LIN {X 0,Y 439.389,Z 296.378,A -85,B 0,C 180,E1 -8958.743,E2 -8958.743} C_VEL
LIN {X 0,Y 439.369,Z 296.379,A -85,B 0,C 180,E1 -8961.609,E2 -8961.609} C_VEL
LIN {X 0,Y 439.4,Z 296.377,A -85,B 0,C 180,E1 -8964.844,E2 -8964.844} C_VEL
LIN {X 0,Y 439.373,Z 296.38,A -85,B 0,C 180,E1 -8968.139,E2 -8968.139} C_VEL
LIN {X 0,Y 439.399,Z 296.377,A -85,B 0,C 180,E1 -8971.606,E2 -8971.606} C_VEL
LIN {X 0,Y 439.372,Z 296.374,A -85,B 0,C 180,E1 -8974.413,E2 -8974.413} C_VEL
LIN {X 0,Y 439.364,Z 296.375,A -85,B 0,C 180,E1 -8977.424,E2 -8977.424} C_VEL
LIN {X 0,Y 439.441,Z 296.372,A -85,B 0,C 180,E1 -8980.663,E2 -8980.663} C_VEL
LIN {X 0,Y 439.463,Z 296.365,A -85,B 0,C 180,E1 -8984.224,E2 -8984.224} C_VEL
LIN {X 0,Y 439.484,Z 296.358,A -85,B 0,C 180,E1 -8988.001,E2 -8988.001} C_VEL
LIN {X 0,Y 439.503,Z 296.366,A -85,B 0,C 180,E1 -8991.725,E2 -8991.725} C_VEL
LIN {X 0,Y 439.603,Z 296.341,A -85,B 0,C 180,E1 -8994.495,E2 -8994.495} C_VEL
LIN {X 0,Y 439.635,Z 296.346,A -85,B 0,C 180,E1 -8998.168,E2 -8998.168} C_VEL
LIN {X 0,Y 439.763,Z 296.319,A -85,B 0,C 180,E1 -9000,E2 -9000} C_VEL
LIN {X 0,Y 439.628,Z 296.347,A -85,B 0,C 180,E1 -9002.749,E2 -9002.749} C_VEL
LIN {X 0,Y 439.595,Z 296.344,A -85,B 0,C 180,E1 -9006.425,E2 -9006.425} C_VEL
LIN {X 0,Y 439.497,Z 296.361,A -85,B 0,C 180,E1 -9009.202,E2 -9009.202} C_VEL
LIN {X 0,Y 439.465,Z 296.366,A -85,B 0,C 180,E1 -9012.938,E2 -9012.938} C_VEL
LIN {X 0,Y 439.446,Z 296.36,A -85,B 0,C 180,E1 -9016.348,E2 -9016.348} C_VEL
LIN {X 0,Y 439.402,Z 296.376,A -85,B 0,C 180,E1 -9019.626,E2 -9019.626} C_VEL
LIN {X 0,Y 439.363,Z 296.377,A -85,B 0,C 180,E1 -9022.575,E2 -9022.575} C_VEL
LIN {X 0,Y 439.371,Z 296.374,A -85,B 0,C 180,E1 -9025.587,E2 -9025.587} C_VEL
LIN {X 0,Y 439.396,Z 296.38,A -85,B 0,C 180,E1 -9028.675,E2 -9028.675} C_VEL
LIN {X 0,Y 439.37,Z 296.382,A -85,B 0,C 180,E1 -9032.03,E2 -9032.03} C_VEL
LIN {X 0,Y 439.392,Z 296.38,A -85,B 0,C 180,E1 -9035.34,E2 -9035.34} C_VEL
LIN {X 0,Y 439.368,Z 296.383,A -85,B 0,C 180,E1 -9038.596,E2 -9038.596} C_VEL
LIN {X 0,Y 439.388,Z 296.377,A -85,B 0,C 180,E1 -9041.257,E2 -9041.257} C_VEL
LIN {X 0,Y 439.398,Z 296.371,A -85,B 0,C 180,E1 -9044.73,E2 -9044.73} C_VEL
LIN {X 0,Y 439.405,Z 296.513,A -85,B 0,C 180,E1 -9045.613,E2 -9045.613} C_VEL
LIN {X 0,Y 442.197,Z 307.685,A -85,B 0,C 180,E1 -9048.888,E2 -9048.888} C_VEL
LIN {X 0,Y 445.159,Z 319.506,A -85,B 0,C 180,E1 -9052.127,E2 -9052.127} C_VEL
LIN {X 0,Y 446.738,Z 326.126,A -85,B 0,C 180,E1 -9053.847,E2 -9053.847} C_VEL
LIN {X 0,Y 445.922,Z 334.334,A -85,B 0,C 180,E1 -9055.706,E2 -9055.706} C_VEL
LIN {X 0,Y 444.194,Z 349.593,A -85,B 0,C 180,E1 -9059.055,E2 -9059.055} C_VEL
LIN {X 0,Y 442.682,Z 366.195,A -85,B 0,C 180,E1 -9062.587,E2 -9062.587} C_VEL
LIN {X 0,Y 441.378,Z 382.993,A -85,B 0,C 180,E1 -9066.044,E2 -9066.044} C_VEL
LIN {X 0,Y 441.077,Z 387.978,A -85,B 0,C 180,E1 -9067.06,E2 -9067.06} C_VEL
LIN {X 0,Y 444.313,Z 406.784,A -85,B 0,C 180,E1 -9067.609,E2 -9067.609} C_VEL
LIN {X 0,Y 446.055,Z 420.769,A -85,B 0,C 180,E1 -9068.139,E2 -9068.139} C_VEL
LIN {X 0,Y 445.379,Z 435.92,A -85,B 0,C 180,E1 -9068.78,E2 -9068.78} C_VEL
LIN {X 0,Y 444.458,Z 449.486,A -85,B 0,C 180,E1 -9069.522,E2 -9069.522} C_VEL
LIN {X 0,Y 443.472,Z 462.876,A -85,B 0,C 180,E1 -9070.441,E2 -9070.441} C_VEL
LIN {X 0,Y 442.399,Z 476.497,A -85,B 0,C 180,E1 -9071.595,E2 -9071.595} C_VEL
LIN {X 0,Y 441.444,Z 489.247,A -85,B 0,C 180,E1 -9072.916,E2 -9072.916} C_VEL
LIN {X 0,Y 440.591,Z 500.172,A -85,B 0,C 180,E1 -9074.266,E2 -9074.266} C_VEL
LIN {X 0,Y 439.816,Z 511.139,A -85,B 0,C 180,E1 -9075.896,E2 -9075.896} C_VEL
LIN {X 0,Y 439.272,Z 519.671,A -85,B 0,C 180,E1 -9077.408,E2 -9077.408} C_VEL
LIN {X 0,Y 439.019,Z 526.835,A -85,B 0,C 180,E1 -9078.925,E2 -9078.925} C_VEL
LIN {X 0,Y 438.661,Z 534.097,A -85,B 0,C 180,E1 -9080.781,E2 -9080.781} C_VEL
LIN {X 0,Y 438.597,Z 539.824,A -85,B 0,C 180,E1 -9082.635,E2 -9082.635} C_VEL
LIN {X 0,Y 438.6,Z 544.148,A -85,B 0,C 180,E1 -9084.483,E2 -9084.483} C_VEL
LIN {X 0,Y 438.618,Z 547.18,A -85,B 0,C 180,E1 -9086.325,E2 -9086.325} C_VEL
LIN {X 0,Y 438.595,Z 548.988,A -85,B 0,C 180,E1 -9088.164,E2 -9088.164} C_VEL
LIN {X 0,Y 438.532,Z 549.6,A -85,B 0,C 180,E1 -9090,E2 -9090} C_VEL
LIN {X 0,Y 438.586,Z 548.989,A -85,B 0,C 180,E1 -9091.837,E2 -9091.837} C_VEL
LIN {X 0,Y 438.643,Z 547.187,A -85,B 0,C 180,E1 -9093.675,E2 -9093.675} C_VEL
LIN {X 0,Y 438.639,Z 544.152,A -85,B 0,C 180,E1 -9095.517,E2 -9095.517} C_VEL
LIN {X 0,Y 438.607,Z 539.818,A -85,B 0,C 180,E1 -9097.365,E2 -9097.365} C_VEL
LIN {X 0,Y 438.683,Z 534.095,A -85,B 0,C 180,E1 -9099.219,E2 -9099.219} C_VEL
LIN {X 0,Y 439.041,Z 526.837,A -85,B 0,C 180,E1 -9101.075,E2 -9101.075} C_VEL
LIN {X 0,Y 439.284,Z 519.632,A -85,B 0,C 180,E1 -9102.598,E2 -9102.598} C_VEL
LIN {X 0,Y 439.825,Z 511.129,A -85,B 0,C 180,E1 -9104.104,E2 -9104.104} C_VEL
LIN {X 0,Y 440.431,Z 501.812,A -85,B 0,C 180,E1 -9105.503,E2 -9105.503} C_VEL
LIN {X 0,Y 441.354,Z 490.463,A -85,B 0,C 180,E1 -9106.939,E2 -9106.939} C_VEL
LIN {X 0,Y 442.217,Z 478.837,A -85,B 0,C 180,E1 -9108.174,E2 -9108.174} C_VEL
LIN {X 0,Y 443.281,Z 465.732,A -85,B 0,C 180,E1 -9109.327,E2 -9109.327} C_VEL
LIN {X 0,Y 444.232,Z 453.008,A -85,B 0,C 180,E1 -9110.248,E2 -9110.248} C_VEL
LIN {X 0,Y 445.224,Z 438.12,A -85,B 0,C 180,E1 -9111.107,E2 -9111.107} C_VEL
LIN {X 0,Y 446.061,Z 422.741,A -85,B 0,C 180,E1 -9111.779,E2 -9111.779} C_VEL
LIN {X 0,Y 445.392,Z 415.694,A -85,B 0,C 180,E1 -9112.067,E2 -9112.067} C_VEL
LIN {X 0,Y 443.655,Z 400.689,A -85,B 0,C 180,E1 -9112.565,E2 -9112.565} C_VEL
LIN {X 0,Y 440.811,Z 384.764,A -85,B 0,C 180,E1 -9113.017,E2 -9113.017} C_VEL
LIN {X 0,Y 441.759,Z 369.337,A -85,B 0,C 180,E1 -9116.199,E2 -9116.199} C_VEL
LIN {X 0,Y 443.194,Z 354.719,A -85,B 0,C 180,E1 -9119.445,E2 -9119.445} C_VEL
LIN {X 0,Y 444.848,Z 342.227,A -85,B 0,C 180,E1 -9122.49,E2 -9122.49} C_VEL
LIN {X 0,Y 447.211,Z 331.063,A -85,B 0,C 180,E1 -9125.554,E2 -9125.554} C_VEL
LIN {X 0,Y 447.513,Z 329.378,A -85,B 0,C 180,E1 -9126.081,E2 -9126.081} C_VEL
LIN {X 0,Y 446.545,Z 324.729,A -85,B 0,C 180,E1 -9127.866,E2 -9127.866} C_VEL
LIN {X 0,Y 445.197,Z 319.492,A -85,B 0,C 180,E1 -9130.334,E2 -9130.334} C_VEL
LIN {X 0,Y 444.029,Z 315.439,A -85,B 0,C 180,E1 -9132.891,E2 -9132.891} C_VEL
LIN {X 0,Y 443.498,Z 313.503,A -85,B 0,C 180,E1 -9134.512,E2 -9134.512} C_VEL
LIN {X 0,Y 442.845,Z 311.488,A -85,B 0,C 180,E1 -9136.968,E2 -9136.968} C_VEL
LIN {X 0,Y 442.349,Z 310.332,A -85,B 0,C 180,E1 -9139.696,E2 -9139.696} C_VEL
LIN {X 0,Y 442.022,Z 310.093,A -85,B 0,C 180,E1 -9142.654,E2 -9142.654} C_VEL
LIN {X 0,Y 441.698,Z 310.52,A -85,B 0,C 180,E1 -9145.054,E2 -9145.054} C_VEL
LIN {X 0,Y 441.188,Z 311.719,A -85,B 0,C 180,E1 -9148.286,E2 -9148.286} C_VEL
LIN {X 0,Y 440.867,Z 313.275,A -85,B 0,C 180,E1 -9151.43,E2 -9151.43} C_VEL
LIN {X 0,Y 440.617,Z 315.071,A -85,B 0,C 180,E1 -9154.491,E2 -9154.491} C_VEL
LIN {X 0,Y 440.408,Z 317.208,A -85,B 0,C 180,E1 -9157.754,E2 -9157.754} C_VEL
LIN {X 0,Y 440.22,Z 319.148,A -85,B 0,C 180,E1 -9160.412,E2 -9160.412} C_VEL
LIN {X 0,Y 440.105,Z 320.778,A -85,B 0,C 180,E1 -9162.575,E2 -9162.575} C_VEL
LIN {X 0,Y 445.525,Z 334.754,A -85,B 0,C 180,E1 -9163.565,E2 -9163.565} C_VEL
LIN {X 0,Y 445.75,Z 336.95,A -85,B 0,C 180,E1 -9163.695,E2 -9163.695} C_VEL
LIN {X 0,Y 445.108,Z 349.492,A -85,B 0,C 180,E1 -9164.43,E2 -9164.43} C_VEL
LIN {X 0,Y 444.362,Z 361.649,A -85,B 0,C 180,E1 -9165.342,E2 -9165.342} C_VEL
LIN {X 0,Y 443.551,Z 372.693,A -85,B 0,C 180,E1 -9166.368,E2 -9166.368} C_VEL
LIN {X 0,Y 442.7,Z 383.554,A -85,B 0,C 180,E1 -9167.625,E2 -9167.625} C_VEL
LIN {X 0,Y 441.92,Z 393.206,A -85,B 0,C 180,E1 -9168.998,E2 -9168.998} C_VEL
LIN {X 0,Y 441.307,Z 400.935,A -85,B 0,C 180,E1 -9170.374,E2 -9170.374} C_VEL
LIN {X 0,Y 440.756,Z 407.201,A -85,B 0,C 180,E1 -9171.749,E2 -9171.749} C_VEL
LIN {X 0,Y 440.312,Z 412.208,A -85,B 0,C 180,E1 -9173.125,E2 -9173.125} C_VEL
LIN {X 0,Y 439.832,Z 416.126,A -85,B 0,C 180,E1 -9174.499,E2 -9174.499} C_VEL
LIN {X 0,Y 439.752,Z 418.15,A -85,B 0,C 180,E1 -9175.417,E2 -9175.417} C_VEL
LIN {X 0,Y 439.742,Z 419.744,A -85,B 0,C 180,E1 -9176.335,E2 -9176.335} C_VEL
LIN {X 0,Y 439.548,Z 420.923,A -85,B 0,C 180,E1 -9177.251,E2 -9177.251} C_VEL
LIN {X 0,Y 439.327,Z 422.086,A -85,B 0,C 180,E1 -9179.083,E2 -9179.083} C_VEL
LIN {X 0,Y 439.293,Z 422.079,A -85,B 0,C 180,E1 -9180,E2 -9180} C_VEL
LIN {X 0,Y 439.301,Z 421.639,A -85,B 0,C 180,E1 -9180.917,E2 -9180.917} C_VEL
LIN {X 0,Y 439.155,Z 419.614,A -85,B 0,C 180,E1 -9182.752,E2 -9182.752} C_VEL
LIN {X 0,Y 439.293,Z 416.979,A -85,B 0,C 180,E1 -9184.129,E2 -9184.129} C_VEL
LIN {X 0,Y 439.475,Z 413.358,A -85,B 0,C 180,E1 -9185.506,E2 -9185.506} C_VEL
LIN {X 0,Y 439.772,Z 408.664,A -85,B 0,C 180,E1 -9186.884,E2 -9186.884} C_VEL
LIN {X 0,Y 440.131,Z 401.693,A -85,B 0,C 180,E1 -9188.494,E2 -9188.494} C_VEL
LIN {X 0,Y 440.5,Z 394.142,A -85,B 0,C 180,E1 -9189.876,E2 -9189.876} C_VEL
LIN {X 0,Y 440.906,Z 384.875,A -85,B 0,C 180,E1 -9191.26,E2 -9191.26} C_VEL
LIN {X 0,Y 441.518,Z 375.436,A -85,B 0,C 180,E1 -9192.409,E2 -9192.409} C_VEL
LIN {X 0,Y 442.075,Z 363.806,A -85,B 0,C 180,E1 -9193.562,E2 -9193.562} C_VEL
LIN {X 0,Y 442.644,Z 351.293,A -85,B 0,C 180,E1 -9194.557,E2 -9194.557} C_VEL
LIN {X 0,Y 443.145,Z 338.462,A -85,B 0,C 180,E1 -9195.346,E2 -9195.346} C_VEL
LIN {X 0,Y 443.417,Z 330.363,A -85,B 0,C 180,E1 -9195.749,E2 -9195.749} C_VEL
LIN {X 0,Y 439.904,Z 316.829,A -85,B 0,C 180,E1 -9196.403,E2 -9196.403} C_VEL
LIN {X 0,Y 438.766,Z 312.57,A -85,B 0,C 180,E1 -9196.589,E2 -9196.589} C_VEL
LIN {X 0,Y 438.819,Z 309.161,A -85,B 0,C 180,E1 -9199.654,E2 -9199.654} C_VEL
LIN {X 0,Y 438.808,Z 305.945,A -85,B 0,C 180,E1 -9202.606,E2 -9202.606} C_VEL
LIN {X 0,Y 438.815,Z 302.707,A -85,B 0,C 180,E1 -9205.622,E2 -9205.622} C_VEL
LIN {X 0,Y 438.855,Z 299.441,A -85,B 0,C 180,E1 -9208.714,E2 -9208.714} C_VEL
LIN {X 0,Y 438.863,Z 297.207,A -85,B 0,C 180,E1 -9210.827,E2 -9210.827} C_VEL
LIN {X 0,Y 438.924,Z 296.439,A -85,B 0,C 180,E1 -9211.936,E2 -9211.936} C_VEL
LIN {X 0,Y 439.305,Z 296.391,A -85,B 0,C 180,E1 -9215.323,E2 -9215.323} C_VEL
LIN {X 0,Y 439.385,Z 296.379,A -85,B 0,C 180,E1 -9218.595,E2 -9218.595} C_VEL
LIN {X 0,Y 439.391,Z 296.374,A -85,B 0,C 180,E1 -9221.257,E2 -9221.257} C_VEL
LIN {X 0,Y 439.401,Z 296.375,A -85,B 0,C 180,E1 -9224.729,E2 -9224.729} C_VEL
LIN {X 0,Y 439.342,Z 296.387,A -85,B 0,C 180,E1 -9228.305,E2 -9228.305} C_VEL
LIN {X 0,Y 439.405,Z 296.687,A -85,B 0,C 180,E1 -9228.741,E2 -9228.741} C_VEL
LIN {X 0,Y 439.466,Z 300.718,A -85,B 0,C 180,E1 -9231.593,E2 -9231.593} C_VEL
LIN {X 0,Y 439.393,Z 305.155,A -85,B 0,C 180,E1 -9234.843,E2 -9234.843} C_VEL
LIN {X 0,Y 439.321,Z 309.591,A -85,B 0,C 180,E1 -9238.135,E2 -9238.135} C_VEL
LIN {X 0,Y 439.259,Z 313.984,A -85,B 0,C 180,E1 -9241.315,E2 -9241.315} C_VEL
LIN {X 0,Y 439.204,Z 318.505,A -85,B 0,C 180,E1 -9244.402,E2 -9244.402} C_VEL
LIN {X 0,Y 439.232,Z 322.302,A -85,B 0,C 180,E1 -9246.82,E2 -9246.82} C_VEL
LIN {X 0,Y 445.434,Z 339.613,A -85,B 0,C 180,E1 -9247.592,E2 -9247.592} C_VEL
LIN {X 0,Y 447.746,Z 347.503,A -85,B 0,C 180,E1 -9247.99,E2 -9247.99} C_VEL
LIN {X 0,Y 447.094,Z 362.755,A -85,B 0,C 180,E1 -9248.636,E2 -9248.636} C_VEL
LIN {X 0,Y 446.37,Z 375.925,A -85,B 0,C 180,E1 -9249.372,E2 -9249.372} C_VEL
LIN {X 0,Y 445.502,Z 389.149,A -85,B 0,C 180,E1 -9250.293,E2 -9250.293} C_VEL
LIN {X 0,Y 444.516,Z 401.345,A -85,B 0,C 180,E1 -9251.327,E2 -9251.327} C_VEL
LIN {X 0,Y 443.447,Z 413.714,A -85,B 0,C 180,E1 -9252.594,E2 -9252.594} C_VEL
LIN {X 0,Y 442.525,Z 424.069,A -85,B 0,C 180,E1 -9253.863,E2 -9253.863} C_VEL
LIN {X 0,Y 441.646,Z 433.644,A -85,B 0,C 180,E1 -9255.249,E2 -9255.249} C_VEL
LIN {X 0,Y 440.798,Z 442.36,A -85,B 0,C 180,E1 -9256.741,E2 -9256.741} C_VEL
LIN {X 0,Y 440.645,Z 444.982,A -85,B 0,C 180,E1 -9257.254,E2 -9257.254} C_VEL
LIN {X 0,Y 439.716,Z 448.238,A -85,B 0,C 180,E1 -9257.885,E2 -9257.885} C_VEL
LIN {X 0,Y 436.468,Z 453.328,A -85,B 0,C 180,E1 -9258.914,E2 -9258.914} C_VEL
LIN {X 0,Y 433.252,Z 457.905,A -85,B 0,C 180,E1 -9259.995,E2 -9259.995} C_VEL
LIN {X 0,Y 432.389,Z 460.347,A -85,B 0,C 180,E1 -9260.699,E2 -9260.699} C_VEL
LIN {X 0,Y 431.991,Z 465.553,A -85,B 0,C 180,E1 -9262.521,E2 -9262.521} C_VEL
LIN {X 0,Y 431.657,Z 469.62,A -85,B 0,C 180,E1 -9264.394,E2 -9264.394} C_VEL
LIN {X 0,Y 431.642,Z 472.459,A -85,B 0,C 180,E1 -9266.266,E2 -9266.266} C_VEL
LIN {X 0,Y 431.424,Z 474.18,A -85,B 0,C 180,E1 -9268.133,E2 -9268.133} C_VEL
LIN {X 0,Y 431.308,Z 474.781,A -85,B 0,C 180,E1 -9270,E2 -9270} C_VEL
LIN {X 0,Y 431.423,Z 474.223,A -85,B 0,C 180,E1 -9271.867,E2 -9271.867} C_VEL
LIN {X 0,Y 431.63,Z 472.562,A -85,B 0,C 180,E1 -9273.734,E2 -9273.734} C_VEL
LIN {X 0,Y 431.653,Z 469.789,A -85,B 0,C 180,E1 -9275.606,E2 -9275.606} C_VEL
LIN {X 0,Y 432.015,Z 465.79,A -85,B 0,C 180,E1 -9277.478,E2 -9277.478} C_VEL
LIN {X 0,Y 432.385,Z 460.486,A -85,B 0,C 180,E1 -9279.354,E2 -9279.354} C_VEL
LIN {X 0,Y 432.988,Z 453.71,A -85,B 0,C 180,E1 -9281.231,E2 -9281.231} C_VEL
LIN {X 0,Y 433.668,Z 446.448,A -85,B 0,C 180,E1 -9282.875,E2 -9282.875} C_VEL
LIN {X 0,Y 434.451,Z 437.686,A -85,B 0,C 180,E1 -9284.521,E2 -9284.521} C_VEL
LIN {X 0,Y 435.515,Z 427.072,A -85,B 0,C 180,E1 -9286.163,E2 -9286.163} C_VEL
LIN {X 0,Y 436.547,Z 416.162,A -85,B 0,C 180,E1 -9287.569,E2 -9287.569} C_VEL
LIN {X 0,Y 437.654,Z 404.17,A -85,B 0,C 180,E1 -9288.855,E2 -9288.855} C_VEL
LIN {X 0,Y 438.74,Z 390.926,A -85,B 0,C 180,E1 -9290.023,E2 -9290.023} C_VEL
LIN {X 0,Y 439.728,Z 377.966,A -85,B 0,C 180,E1 -9290.953,E2 -9290.953} C_VEL
LIN {X 0,Y 440.589,Z 363.194,A -85,B 0,C 180,E1 -9291.797,E2 -9291.797} C_VEL
LIN {X 0,Y 441.033,Z 348.463,A -85,B 0,C 180,E1 -9292.444,E2 -9292.444} C_VEL
LIN {X 0,Y 436.308,Z 334.096,A -85,B 0,C 180,E1 -9293.182,E2 -9293.182} C_VEL
LIN {X 0,Y 432.227,Z 322.877,A -85,B 0,C 180,E1 -9293.677,E2 -9293.677} C_VEL
LIN {X 0,Y 432.245,Z 317.598,A -85,B 0,C 180,E1 -9297.082,E2 -9297.082} C_VEL
LIN {X 0,Y 432.289,Z 313.042,A -85,B 0,C 180,E1 -9300.264,E2 -9300.264} C_VEL
LIN {X 0,Y 432.357,Z 307.993,A -85,B 0,C 180,E1 -9304.003,E2 -9304.003} C_VEL
LIN {X 0,Y 432.41,Z 303.622,A -85,B 0,C 180,E1 -9307.212,E2 -9307.212} C_VEL
LIN {X 0,Y 432.456,Z 299.531,A -85,B 0,C 180,E1 -9310.198,E2 -9310.198} C_VEL
LIN {X 0,Y 432.31,Z 297.266,A -85,B 0,C 180,E1 -9311.8,E2 -9311.8} C_VEL
LIN {X 0,Y 432.333,Z 297.26,A -85,B 0,C 180,E1 -9314.347,E2 -9314.347} C_VEL
LIN {X 0,Y 432.321,Z 297.262,A -85,B 0,C 180,E1 -9317.015,E2 -9317.015} C_VEL
LIN {X 0,Y 432.333,Z 297.258,A -85,B 0,C 180,E1 -9319.821,E2 -9319.821} C_VEL
LIN {X 0,Y 432.306,Z 297.26,A -85,B 0,C 180,E1 -9323.022,E2 -9323.022} C_VEL
LIN {X 0,Y 432.36,Z 297.25,A -85,B 0,C 180,E1 -9325.996,E2 -9325.996} C_VEL
LIN {X 0,Y 432.346,Z 297.251,A -85,B 0,C 180,E1 -9329.49,E2 -9329.49} C_VEL
LIN {X 0,Y 432.327,Z 297.26,A -85,B 0,C 180,E1 -9331.873,E2 -9331.873} C_VEL
LIN {X 0,Y 432.376,Z 297.253,A -85,B 0,C 180,E1 -9335.539,E2 -9335.539} C_VEL
LIN {X 0,Y 432.35,Z 297.251,A -85,B 0,C 180,E1 -9339.046,E2 -9339.046} C_VEL
LIN {X 0,Y 432.358,Z 297.249,A -85,B 0,C 180,E1 -9342.01,E2 -9342.01} C_VEL
LIN {X 0,Y 432.397,Z 297.247,A -85,B 0,C 180,E1 -9344.926,E2 -9344.926} C_VEL
LIN {X 0,Y 432.46,Z 297.232,A -85,B 0,C 180,E1 -9347.803,E2 -9347.803} C_VEL
LIN {X 0,Y 432.463,Z 297.242,A -85,B 0,C 180,E1 -9351.59,E2 -9351.59} C_VEL
LIN {X 0,Y 432.576,Z 297.215,A -85,B 0,C 180,E1 -9354.406,E2 -9354.406} C_VEL
LIN {X 0,Y 432.604,Z 297.221,A -85,B 0,C 180,E1 -9358.138,E2 -9358.138} C_VEL
LIN {X 0,Y 432.733,Z 297.194,A -85,B 0,C 180,E1 -9360,E2 -9360} C_VEL
LIN {X 0,Y 432.579,Z 297.225,A -85,B 0,C 180,E1 -9362.794,E2 -9362.794} C_VEL
LIN {X 0,Y 432.547,Z 297.223,A -85,B 0,C 180,E1 -9366.531,E2 -9366.531} C_VEL
LIN {X 0,Y 432.441,Z 297.24,A -85,B 0,C 180,E1 -9369.353,E2 -9369.353} C_VEL
LIN {X 0,Y 432.431,Z 297.242,A -85,B 0,C 180,E1 -9372.803,E2 -9372.803} C_VEL
LIN {X 0,Y 432.411,Z 297.236,A -85,B 0,C 180,E1 -9376.478,E2 -9376.478} C_VEL
LIN {X 0,Y 432.339,Z 297.258,A -85,B 0,C 180,E1 -9379.96,E2 -9379.96} C_VEL
LIN {X 0,Y 432.316,Z 297.255,A -85,B 0,C 180,E1 -9382.964,E2 -9382.964} C_VEL
LIN {X 0,Y 432.333,Z 297.258,A -85,B 0,C 180,E1 -9385.002,E2 -9385.002} C_VEL
LIN {X 0,Y 432.342,Z 297.253,A -85,B 0,C 180,E1 -9388.126,E2 -9388.126} C_VEL
LIN {X 0,Y 432.32,Z 297.258,A -85,B 0,C 180,E1 -9391.346,E2 -9391.346} C_VEL
LIN {X 0,Y 432.338,Z 297.255,A -85,B 0,C 180,E1 -9394.677,E2 -9394.677} C_VEL
LIN {X 0,Y 432.331,Z 297.259,A -85,B 0,C 180,E1 -9398.15,E2 -9398.15} C_VEL
LIN {X 0,Y 432.332,Z 297.256,A -85,B 0,C 180,E1 -9401.602,E2 -9401.602} C_VEL
LIN {X 0,Y 432.369,Z 297.359,A -85,B 0,C 180,E1 -9405.08,E2 -9405.08} C_VEL
LIN {X 0,Y 435.202,Z 308.884,A -85,B 0,C 180,E1 -9408.54,E2 -9408.54} C_VEL
LIN {X 0,Y 437.783,Z 319.165,A -85,B 0,C 180,E1 -9411.427,E2 -9411.427} C_VEL
LIN {X 0,Y 439.885,Z 327.94,A -85,B 0,C 180,E1 -9413.762,E2 -9413.762} C_VEL
LIN {X 0,Y 439.027,Z 336.115,A -85,B 0,C 180,E1 -9415.647,E2 -9415.647} C_VEL
LIN {X 0,Y 437.106,Z 352.498,A -85,B 0,C 180,E1 -9419.304,E2 -9419.304} C_VEL
LIN {X 0,Y 435.528,Z 368.731,A -85,B 0,C 180,E1 -9422.825,E2 -9422.825} C_VEL
LIN {X 0,Y 434.297,Z 384.479,A -85,B 0,C 180,E1 -9426.136,E2 -9426.136} C_VEL
LIN {X 0,Y 434.111,Z 387.031,A -85,B 0,C 180,E1 -9426.663,E2 -9426.663} C_VEL
LIN {X 0,Y 437.608,Z 406.962,A -85,B 0,C 180,E1 -9427.267,E2 -9427.267} C_VEL
LIN {X 0,Y 439.369,Z 421.804,A -85,B 0,C 180,E1 -9427.854,E2 -9427.854} C_VEL
LIN {X 0,Y 438.658,Z 436.472,A -85,B 0,C 180,E1 -9428.501,E2 -9428.501} C_VEL
LIN {X 0,Y 437.619,Z 450.671,A -85,B 0,C 180,E1 -9429.31,E2 -9429.31} C_VEL
LIN {X 0,Y 436.582,Z 463.723,A -85,B 0,C 180,E1 -9430.242,E2 -9430.242} C_VEL
LIN {X 0,Y 435.473,Z 477.078,A -85,B 0,C 180,E1 -9431.413,E2 -9431.413} C_VEL
LIN {X 0,Y 434.589,Z 488.148,A -85,B 0,C 180,E1 -9432.578,E2 -9432.578} C_VEL
LIN {X 0,Y 433.658,Z 499.56,A -85,B 0,C 180,E1 -9434.008,E2 -9434.008} C_VEL
LIN {X 0,Y 432.803,Z 510.523,A -85,B 0,C 180,E1 -9435.663,E2 -9435.663} C_VEL
LIN {X 0,Y 432.21,Z 519.683,A -85,B 0,C 180,E1 -9437.326,E2 -9437.326} C_VEL
LIN {X 0,Y 431.875,Z 528.205,A -85,B 0,C 180,E1 -9439.214,E2 -9439.214} C_VEL
LIN {X 0,Y 431.551,Z 535.064,A -85,B 0,C 180,E1 -9441.1,E2 -9441.1} C_VEL
LIN {X 0,Y 431.515,Z 540.444,A -85,B 0,C 180,E1 -9442.984,E2 -9442.984} C_VEL
LIN {X 0,Y 431.533,Z 543.539,A -85,B 0,C 180,E1 -9444.392,E2 -9444.392} C_VEL
LIN {X 0,Y 431.549,Z 546.572,A -85,B 0,C 180,E1 -9446.265,E2 -9446.265} C_VEL
LIN {X 0,Y 431.533,Z 548.38,A -85,B 0,C 180,E1 -9448.134,E2 -9448.134} C_VEL
LIN {X 0,Y 431.461,Z 548.992,A -85,B 0,C 180,E1 -9450,E2 -9450} C_VEL
LIN {X 0,Y 431.525,Z 548.382,A -85,B 0,C 180,E1 -9451.867,E2 -9451.867} C_VEL
LIN {X 0,Y 431.577,Z 546.578,A -85,B 0,C 180,E1 -9453.735,E2 -9453.735} C_VEL
LIN {X 0,Y 431.57,Z 543.541,A -85,B 0,C 180,E1 -9455.607,E2 -9455.607} C_VEL
LIN {X 0,Y 431.527,Z 539.204,A -85,B 0,C 180,E1 -9457.487,E2 -9457.487} C_VEL
LIN {X 0,Y 431.621,Z 533.48,A -85,B 0,C 180,E1 -9459.371,E2 -9459.371} C_VEL
LIN {X 0,Y 431.949,Z 526.217,A -85,B 0,C 180,E1 -9461.259,E2 -9461.259} C_VEL
LIN {X 0,Y 432.27,Z 519.036,A -85,B 0,C 180,E1 -9462.802,E2 -9462.802} C_VEL
LIN {X 0,Y 432.813,Z 510.509,A -85,B 0,C 180,E1 -9464.337,E2 -9464.337} C_VEL
LIN {X 0,Y 433.514,Z 501.198,A -85,B 0,C 180,E1 -9465.757,E2 -9465.757} C_VEL
LIN {X 0,Y 434.402,Z 490.739,A -85,B 0,C 180,E1 -9467.11,E2 -9467.11} C_VEL
LIN {X 0,Y 435.281,Z 479.413,A -85,B 0,C 180,E1 -9468.352,E2 -9468.352} C_VEL
LIN {X 0,Y 436.39,Z 466.562,A -85,B 0,C 180,E1 -9469.523,E2 -9469.523} C_VEL
LIN {X 0,Y 437.509,Z 452.406,A -85,B 0,C 180,E1 -9470.573,E2 -9470.573} C_VEL
LIN {X 0,Y 438.566,Z 437.529,A -85,B 0,C 180,E1 -9471.443,E2 -9471.443} C_VEL
LIN {X 0,Y 439.406,Z 422.466,A -85,B 0,C 180,E1 -9472.113,E2 -9472.113} C_VEL
LIN {X 0,Y 438.021,Z 409.096,A -85,B 0,C 180,E1 -9472.649,E2 -9472.649} C_VEL
LIN {X 0,Y 435.807,Z 394.15,A -85,B 0,C 180,E1 -9473.114,E2 -9473.114} C_VEL
LIN {X 0,Y 433.881,Z 384.095,A -85,B 0,C 180,E1 -9473.4,E2 -9473.4} C_VEL
LIN {X 0,Y 434.835,Z 370.016,A -85,B 0,C 180,E1 -9476.39,E2 -9476.39} C_VEL
LIN {X 0,Y 436.288,Z 356.108,A -85,B 0,C 180,E1 -9479.557,E2 -9479.557} C_VEL
LIN {X 0,Y 437.947,Z 344.254,A -85,B 0,C 180,E1 -9482.52,E2 -9482.52} C_VEL
LIN {X 0,Y 440.259,Z 333.601,A -85,B 0,C 180,E1 -9485.499,E2 -9485.499} C_VEL
LIN {X 0,Y 440.73,Z 331.477,A -85,B 0,C 180,E1 -9486.158,E2 -9486.158} C_VEL
LIN {X 0,Y 439.842,Z 327.067,A -85,B 0,C 180,E1 -9487.883,E2 -9487.883} C_VEL
LIN {X 0,Y 438.472,Z 321.694,A -85,B 0,C 180,E1 -9490.455,E2 -9490.455} C_VEL
LIN {X 0,Y 437.565,Z 318.506,A -85,B 0,C 180,E1 -9492.423,E2 -9492.423} C_VEL
LIN {X 0,Y 436.63,Z 315.319,A -85,B 0,C 180,E1 -9495.091,E2 -9495.091} C_VEL
LIN {X 0,Y 435.941,Z 313.273,A -85,B 0,C 180,E1 -9497.867,E2 -9497.867} C_VEL
LIN {X 0,Y 435.452,Z 312.288,A -85,B 0,C 180,E1 -9500.778,E2 -9500.778} C_VEL
LIN {X 0,Y 435.131,Z 312.192,A -85,B 0,C 180,E1 -9503.302,E2 -9503.302} C_VEL
LIN {X 0,Y 434.789,Z 312.607,A -85,B 0,C 180,E1 -9505.546,E2 -9505.546} C_VEL
LIN {X 0,Y 434.246,Z 313.864,A -85,B 0,C 180,E1 -9509.068,E2 -9509.068} C_VEL
LIN {X 0,Y 433.907,Z 315.279,A -85,B 0,C 180,E1 -9511.984,E2 -9511.984} C_VEL
LIN {X 0,Y 433.654,Z 317.108,A -85,B 0,C 180,E1 -9515.171,E2 -9515.171} C_VEL
LIN {X 0,Y 433.449,Z 319.023,A -85,B 0,C 180,E1 -9518.104,E2 -9518.104} C_VEL
LIN {X 0,Y 433.236,Z 321.149,A -85,B 0,C 180,E1 -9521.068,E2 -9521.068} C_VEL
LIN {X 0,Y 433.204,Z 322.098,A -85,B 0,C 180,E1 -9522.151,E2 -9522.151} C_VEL
LIN {X 0,Y 438.344,Z 334.617,A -85,B 0,C 180,E1 -9523.078,E2 -9523.078} C_VEL
LIN {X 0,Y 439.309,Z 337.522,A -85,B 0,C 180,E1 -9523.303,E2 -9523.303} C_VEL
LIN {X 0,Y 438.617,Z 350.508,A -85,B 0,C 180,E1 -9524.084,E2 -9524.084} C_VEL
LIN {X 0,Y 437.701,Z 363.845,A -85,B 0,C 180,E1 -9525.114,E2 -9525.114} C_VEL
LIN {X 0,Y 436.891,Z 374.635,A -85,B 0,C 180,E1 -9526.156,E2 -9526.156} C_VEL
LIN {X 0,Y 435.986,Z 385.314,A -85,B 0,C 180,E1 -9527.431,E2 -9527.431} C_VEL
LIN {X 0,Y 435.115,Z 394.767,A -85,B 0,C 180,E1 -9528.824,E2 -9528.824} C_VEL
LIN {X 0,Y 434.31,Z 403.527,A -85,B 0,C 180,E1 -9530.453,E2 -9530.453} C_VEL
LIN {X 0,Y 433.868,Z 408.59,A -85,B 0,C 180,E1 -9531.617,E2 -9531.617} C_VEL
LIN {X 0,Y 433.399,Z 413.543,A -85,B 0,C 180,E1 -9533.015,E2 -9533.015} C_VEL
LIN {X 0,Y 432.882,Z 417.409,A -85,B 0,C 180,E1 -9534.41,E2 -9534.41} C_VEL
LIN {X 0,Y 432.794,Z 419.388,A -85,B 0,C 180,E1 -9535.343,E2 -9535.343} C_VEL
LIN {X 0,Y 432.757,Z 420.935,A -85,B 0,C 180,E1 -9536.276,E2 -9536.276} C_VEL
LIN {X 0,Y 432.381,Z 422.822,A -85,B 0,C 180,E1 -9538.137,E2 -9538.137} C_VEL
LIN {X 0,Y 432.313,Z 423.181,A -85,B 0,C 180,E1 -9539.069,E2 -9539.069} C_VEL
LIN {X 0,Y 432.274,Z 423.143,A -85,B 0,C 180,E1 -9540,E2 -9540} C_VEL
LIN {X 0,Y 432.281,Z 422.672,A -85,B 0,C 180,E1 -9540.932,E2 -9540.932} C_VEL
LIN {X 0,Y 432.129,Z 420.581,A -85,B 0,C 180,E1 -9542.797,E2 -9542.797} C_VEL
LIN {X 0,Y 432.278,Z 417.89,A -85,B 0,C 180,E1 -9544.196,E2 -9544.196} C_VEL
LIN {X 0,Y 432.478,Z 414.213,A -85,B 0,C 180,E1 -9545.596,E2 -9545.596} C_VEL
LIN {X 0,Y 432.782,Z 409.459,A -85,B 0,C 180,E1 -9546.996,E2 -9546.996} C_VEL
LIN {X 0,Y 433.146,Z 402.399,A -85,B 0,C 180,E1 -9548.632,E2 -9548.632} C_VEL
LIN {X 0,Y 433.554,Z 394.776,A -85,B 0,C 180,E1 -9550.036,E2 -9550.036} C_VEL
LIN {X 0,Y 433.965,Z 385.428,A -85,B 0,C 180,E1 -9551.443,E2 -9551.443} C_VEL
LIN {X 0,Y 434.685,Z 374.809,A -85,B 0,C 180,E1 -9552.726,E2 -9552.726} C_VEL
LIN {X 0,Y 435.27,Z 362.872,A -85,B 0,C 180,E1 -9553.897,E2 -9553.897} C_VEL
LIN {X 0,Y 435.839,Z 350.436,A -85,B 0,C 180,E1 -9554.865,E2 -9554.865} C_VEL
LIN {X 0,Y 436.379,Z 337.522,A -85,B 0,C 180,E1 -9555.65,E2 -9555.65} C_VEL
LIN {X 0,Y 436.556,Z 331.561,A -85,B 0,C 180,E1 -9555.948,E2 -9555.948} C_VEL
LIN {X 0,Y 432.936,Z 317.83,A -85,B 0,C 180,E1 -9556.637,E2 -9556.637} C_VEL
LIN {X 0,Y 431.731,Z 313.107,A -85,B 0,C 180,E1 -9556.85,E2 -9556.85} C_VEL
LIN {X 0,Y 431.755,Z 309.621,A -85,B 0,C 180,E1 -9559.989,E2 -9559.989} C_VEL
LIN {X 0,Y 431.76,Z 306.364,A -85,B 0,C 180,E1 -9562.996,E2 -9562.996} C_VEL
LIN {X 0,Y 431.771,Z 303.043,A -85,B 0,C 180,E1 -9566.071,E2 -9566.071} C_VEL
LIN {X 0,Y 431.811,Z 299.714,A -85,B 0,C 180,E1 -9569.227,E2 -9569.227} C_VEL
LIN {X 0,Y 431.826,Z 297.447,A -85,B 0,C 180,E1 -9571.386,E2 -9571.386} C_VEL
LIN {X 0,Y 432.192,Z 297.274,A -85,B 0,C 180,E1 -9574.691,E2 -9574.691} C_VEL
LIN {X 0,Y 432.339,Z 297.254,A -85,B 0,C 180,E1 -9578.15,E2 -9578.15} C_VEL
LIN {X 0,Y 432.335,Z 297.252,A -85,B 0,C 180,E1 -9581.602,E2 -9581.602} C_VEL
LIN {X 0,Y 432.336,Z 297.255,A -85,B 0,C 180,E1 -9584.347,E2 -9584.347} C_VEL
LIN {X 0,Y 432.301,Z 297.262,A -85,B 0,C 180,E1 -9587.019,E2 -9587.019} C_VEL
LIN {X 0,Y 432.326,Z 297.377,A -85,B 0,C 180,E1 -9588.399,E2 -9588.399} C_VEL
LIN {X 0,Y 432.427,Z 300.564,A -85,B 0,C 180,E1 -9590.665,E2 -9590.665} C_VEL
LIN {X 0,Y 432.396,Z 303.811,A -85,B 0,C 180,E1 -9593.031,E2 -9593.031} C_VEL
LIN {X 0,Y 432.33,Z 308.417,A -85,B 0,C 180,E1 -9596.447,E2 -9596.447} C_VEL
LIN {X 0,Y 432.284,Z 312.899,A -85,B 0,C 180,E1 -9599.735,E2 -9599.735} C_VEL
LIN {X 0,Y 432.222,Z 317.438,A -85,B 0,C 180,E1 -9602.916,E2 -9602.916} C_VEL
LIN {X 0,Y 432.212,Z 322.882,A -85,B 0,C 180,E1 -9606.428,E2 -9606.428} C_VEL
LIN {X 0,Y 438.221,Z 339.405,A -85,B 0,C 180,E1 -9607.179,E2 -9607.179} C_VEL
LIN {X 0,Y 441.132,Z 349.115,A -85,B 0,C 180,E1 -9607.681,E2 -9607.681} C_VEL
LIN {X 0,Y 440.511,Z 363.658,A -85,B 0,C 180,E1 -9608.317,E2 -9608.317} C_VEL
LIN {X 0,Y 439.775,Z 376.516,A -85,B 0,C 180,E1 -9609.049,E2 -9609.049} C_VEL
LIN {X 0,Y 438.866,Z 389.745,A -85,B 0,C 180,E1 -9609.983,E2 -9609.983} C_VEL
LIN {X 0,Y 437.805,Z 401.947,A -85,B 0,C 180,E1 -9611.03,E2 -9611.03} C_VEL
LIN {X 0,Y 436.699,Z 414.318,A -85,B 0,C 180,E1 -9612.316,E2 -9612.316} C_VEL
LIN {X 0,Y 435.748,Z 424.673,A -85,B 0,C 180,E1 -9613.605,E2 -9613.605} C_VEL
LIN {X 0,Y 434.811,Z 434.25,A -85,B 0,C 180,E1 -9615.012,E2 -9615.012} C_VEL
LIN {X 0,Y 433.868,Z 443.238,A -85,B 0,C 180,E1 -9616.579,E2 -9616.579} C_VEL
LIN {X 0,Y 433.188,Z 451.387,A -85,B 0,C 180,E1 -9618.299,E2 -9618.299} C_VEL
LIN {X 0,Y 432.531,Z 458.625,A -85,B 0,C 180,E1 -9620.176,E2 -9620.176} C_VEL
LIN {X 0,Y 432.389,Z 460.347,A -85,B 0,C 180,E1 -9620.699,E2 -9620.699} C_VEL
LIN {X 0,Y 431.534,Z 462.652,A -85,B 0,C 180,E1 -9621.414,E2 -9621.414} C_VEL
LIN {X 0,Y 427.001,Z 467.444,A -85,B 0,C 180,E1 -9623.049,E2 -9623.049} C_VEL
LIN {X 0,Y 424.936,Z 469.714,A -85,B 0,C 180,E1 -9624.033,E2 -9624.033} C_VEL
LIN {X 0,Y 424.602,Z 470.637,A -85,B 0,C 180,E1 -9624.549,E2 -9624.549} C_VEL
LIN {X 0,Y 424.579,Z 473.068,A -85,B 0,C 180,E1 -9626.203,E2 -9626.203} C_VEL
LIN {X 0,Y 424.373,Z 474.787,A -85,B 0,C 180,E1 -9628.102,E2 -9628.102} C_VEL
LIN {X 0,Y 424.248,Z 475.389,A -85,B 0,C 180,E1 -9630,E2 -9630} C_VEL
LIN {X 0,Y 424.372,Z 474.83,A -85,B 0,C 180,E1 -9631.898,E2 -9631.898} C_VEL
LIN {X 0,Y 424.569,Z 473.17,A -85,B 0,C 180,E1 -9633.796,E2 -9633.796} C_VEL
LIN {X 0,Y 424.604,Z 470.397,A -85,B 0,C 180,E1 -9635.699,E2 -9635.699} C_VEL
LIN {X 0,Y 424.99,Z 466.398,A -85,B 0,C 180,E1 -9637.602,E2 -9637.602} C_VEL
LIN {X 0,Y 425.394,Z 461.092,A -85,B 0,C 180,E1 -9639.509,E2 -9639.509} C_VEL
LIN {X 0,Y 426.049,Z 454.314,A -85,B 0,C 180,E1 -9641.417,E2 -9641.417} C_VEL
LIN {X 0,Y 426.762,Z 447.052,A -85,B 0,C 180,E1 -9643.087,E2 -9643.087} C_VEL
LIN {X 0,Y 427.588,Z 438.289,A -85,B 0,C 180,E1 -9644.759,E2 -9644.759} C_VEL
LIN {X 0,Y 428.704,Z 427.673,A -85,B 0,C 180,E1 -9646.427,E2 -9646.427} C_VEL
LIN {X 0,Y 429.778,Z 416.761,A -85,B 0,C 180,E1 -9647.855,E2 -9647.855} C_VEL
LIN {X 0,Y 430.964,Z 404.762,A -85,B 0,C 180,E1 -9649.159,E2 -9649.159} C_VEL
LIN {X 0,Y 432.105,Z 391.511,A -85,B 0,C 180,E1 -9650.344,E2 -9650.344} C_VEL
LIN {X 0,Y 433.138,Z 378.545,A -85,B 0,C 180,E1 -9651.288,E2 -9651.288} C_VEL
LIN {X 0,Y 434.022,Z 364.224,A -85,B 0,C 180,E1 -9652.12,E2 -9652.12} C_VEL
LIN {X 0,Y 434.513,Z 350.164,A -85,B 0,C 180,E1 -9652.754,E2 -9652.754} C_VEL
LIN {X 0,Y 429.898,Z 336.047,A -85,B 0,C 180,E1 -9653.507,E2 -9653.507} C_VEL
LIN {X 0,Y 425.205,Z 323.442,A -85,B 0,C 180,E1 -9654.095,E2 -9654.095} C_VEL
LIN {X 0,Y 425.231,Z 318.071,A -85,B 0,C 180,E1 -9657.566,E2 -9657.566} C_VEL
LIN {X 0,Y 425.271,Z 314.997,A -85,B 0,C 180,E1 -9659.721,E2 -9659.721} C_VEL
LIN {X 0,Y 425.291,Z 310.392,A -85,B 0,C 180,E1 -9663.047,E2 -9663.047} C_VEL
LIN {X 0,Y 425.339,Z 306.513,A -85,B 0,C 180,E1 -9665.939,E2 -9665.939} C_VEL
LIN {X 0,Y 425.44,Z 302.256,A -85,B 0,C 180,E1 -9669.067,E2 -9669.067} C_VEL
LIN {X 0,Y 425.374,Z 299.058,A -85,B 0,C 180,E1 -9671.367,E2 -9671.367} C_VEL
LIN {X 0,Y 425.256,Z 298.143,A -85,B 0,C 180,E1 -9672.07,E2 -9672.07} C_VEL
LIN {X 0,Y 425.285,Z 298.14,A -85,B 0,C 180,E1 -9675.283,E2 -9675.283} C_VEL
LIN {X 0,Y 425.274,Z 298.136,A -85,B 0,C 180,E1 -9678.621,E2 -9678.621} C_VEL
LIN {X 0,Y 425.292,Z 298.131,A -85,B 0,C 180,E1 -9681.101,E2 -9681.101} C_VEL
LIN {X 0,Y 425.3,Z 298.133,A -85,B 0,C 180,E1 -9684.664,E2 -9684.664} C_VEL
LIN {X 0,Y 425.265,Z 298.137,A -85,B 0,C 180,E1 -9688.073,E2 -9688.073} C_VEL
LIN {X 0,Y 425.304,Z 298.131,A -85,B 0,C 180,E1 -9691.366,E2 -9691.366} C_VEL
LIN {X 0,Y 425.266,Z 298.131,A -85,B 0,C 180,E1 -9694.553,E2 -9694.553} C_VEL
LIN {X 0,Y 425.304,Z 298.134,A -85,B 0,C 180,E1 -9696.635,E2 -9696.635} C_VEL
LIN {X 0,Y 425.328,Z 298.132,A -85,B 0,C 180,E1 -9700.365,E2 -9700.365} C_VEL
LIN {X 0,Y 425.387,Z 298.113,A -85,B 0,C 180,E1 -9703.688,E2 -9703.688} C_VEL
LIN {X 0,Y 425.413,Z 298.11,A -85,B 0,C 180,E1 -9707.598,E2 -9707.598} C_VEL
LIN {X 0,Y 425.408,Z 298.12,A -85,B 0,C 180,E1 -9711.449,E2 -9711.449} C_VEL
LIN {X 0,Y 425.531,Z 298.093,A -85,B 0,C 180,E1 -9714.313,E2 -9714.313} C_VEL
LIN {X 0,Y 425.574,Z 298.097,A -85,B 0,C 180,E1 -9718.107,E2 -9718.107} C_VEL
LIN {X 0,Y 425.702,Z 298.07,A -85,B 0,C 180,E1 -9720,E2 -9720} C_VEL
LIN {X 0,Y 425.533,Z 298.103,A -85,B 0,C 180,E1 -9722.84,E2 -9722.84} C_VEL
LIN {X 0,Y 425.536,Z 298.092,A -85,B 0,C 180,E1 -9725.687,E2 -9725.687} C_VEL
LIN {X 0,Y 425.409,Z 298.121,A -85,B 0,C 180,E1 -9728.551,E2 -9728.551} C_VEL
LIN {X 0,Y 425.412,Z 298.117,A -85,B 0,C 180,E1 -9732.402,E2 -9732.402} C_VEL
LIN {X 0,Y 425.387,Z 298.11,A -85,B 0,C 180,E1 -9736.312,E2 -9736.312} C_VEL
LIN {X 0,Y 425.328,Z 298.129,A -85,B 0,C 180,E1 -9739.635,E2 -9739.635} C_VEL
LIN {X 0,Y 425.287,Z 298.128,A -85,B 0,C 180,E1 -9742.339,E2 -9742.339} C_VEL
LIN {X 0,Y 425.316,Z 298.131,A -85,B 0,C 180,E1 -9744.656,E2 -9744.656} C_VEL
LIN {X 0,Y 425.268,Z 298.133,A -85,B 0,C 180,E1 -9747.563,E2 -9747.563} C_VEL
LIN {X 0,Y 425.29,Z 298.134,A -85,B 0,C 180,E1 -9750.761,E2 -9750.761} C_VEL
LIN {X 0,Y 425.31,Z 298.13,A -85,B 0,C 180,E1 -9754.288,E2 -9754.288} C_VEL
LIN {X 0,Y 425.275,Z 298.136,A -85,B 0,C 180,E1 -9757.695,E2 -9757.695} C_VEL
LIN {X 0,Y 425.279,Z 298.136,A -85,B 0,C 180,E1 -9760.52,E2 -9760.52} C_VEL
LIN {X 0,Y 425.256,Z 298.133,A -85,B 0,C 180,E1 -9763.351,E2 -9763.351} C_VEL
LIN {X 0,Y 425.344,Z 298.272,A -85,B 0,C 180,E1 -9764.566,E2 -9764.566} C_VEL
LIN {X 0,Y 428.329,Z 310.442,A -85,B 0,C 180,E1 -9768.293,E2 -9768.293} C_VEL
LIN {X 0,Y 431.108,Z 321.617,A -85,B 0,C 180,E1 -9771.49,E2 -9771.49} C_VEL
LIN {X 0,Y 433.048,Z 329.714,A -85,B 0,C 180,E1 -9773.675,E2 -9773.675} C_VEL
LIN {X 0,Y 431.653,Z 341.315,A -85,B 0,C 180,E1 -9776.388,E2 -9776.388} C_VEL
LIN {X 0,Y 429.699,Z 357.753,A -85,B 0,C 180,E1 -9780.094,E2 -9780.094} C_VEL
LIN {X 0,Y 428.327,Z 371.783,A -85,B 0,C 180,E1 -9783.178,E2 -9783.178} C_VEL
LIN {X 0,Y 427.18,Z 386.052,A -85,B 0,C 180,E1 -9786.251,E2 -9786.251} C_VEL
LIN {X 0,Y 430.841,Z 406.697,A -85,B 0,C 180,E1 -9786.897,E2 -9786.897} C_VEL
LIN {X 0,Y 432.586,Z 422.425,A -85,B 0,C 180,E1 -9787.537,E2 -9787.537} C_VEL
LIN {X 0,Y 432.342,Z 430.375,A -85,B 0,C 180,E1 -9787.884,E2 -9787.884} C_VEL
LIN {X 0,Y 431.359,Z 444.625,A -85,B 0,C 180,E1 -9788.634,E2 -9788.634} C_VEL
LIN {X 0,Y 430.225,Z 458.515,A -85,B 0,C 180,E1 -9789.563,E2 -9789.563} C_VEL
LIN {X 0,Y 429.121,Z 471.428,A -85,B 0,C 180,E1 -9790.631,E2 -9790.631} C_VEL
LIN {X 0,Y 428.057,Z 483.371,A -85,B 0,C 180,E1 -9791.823,E2 -9791.823} C_VEL
LIN {X 0,Y 426.998,Z 495.351,A -85,B 0,C 180,E1 -9793.26,E2 -9793.26} C_VEL
LIN {X 0,Y 426.144,Z 505.437,A -85,B 0,C 180,E1 -9794.7,E2 -9794.7} C_VEL
LIN {X 0,Y 425.464,Z 515.309,A -85,B 0,C 180,E1 -9796.386,E2 -9796.386} C_VEL
LIN {X 0,Y 424.948,Z 523.535,A -85,B 0,C 180,E1 -9798.069,E2 -9798.069} C_VEL
LIN {X 0,Y 424.68,Z 529.441,A -85,B 0,C 180,E1 -9799.512,E2 -9799.512} C_VEL
LIN {X 0,Y 424.468,Z 535.918,A -85,B 0,C 180,E1 -9801.43,E2 -9801.43} C_VEL
LIN {X 0,Y 424.44,Z 541.2,A -85,B 0,C 180,E1 -9803.461,E2 -9803.461} C_VEL
LIN {X 0,Y 424.379,Z 544.594,A -85,B 0,C 180,E1 -9805.25,E2 -9805.25} C_VEL
LIN {X 0,Y 424.5,Z 547.02,A -85,B 0,C 180,E1 -9807.153,E2 -9807.153} C_VEL
LIN {X 0,Y 424.402,Z 548.226,A -85,B 0,C 180,E1 -9809.051,E2 -9809.051} C_VEL
LIN {X 0,Y 424.401,Z 548.227,A -85,B 0,C 180,E1 -9810.949,E2 -9810.949} C_VEL
LIN {X 0,Y 424.508,Z 547.023,A -85,B 0,C 180,E1 -9812.847,E2 -9812.847} C_VEL
LIN {X 0,Y 424.445,Z 544.602,A -85,B 0,C 180,E1 -9814.749,E2 -9814.749} C_VEL
LIN {X 0,Y 424.498,Z 540.93,A -85,B 0,C 180,E1 -9816.655,E2 -9816.655} C_VEL
LIN {X 0,Y 424.476,Z 535.909,A -85,B 0,C 180,E1 -9818.57,E2 -9818.57} C_VEL
LIN {X 0,Y 424.704,Z 529.438,A -85,B 0,C 180,E1 -9820.488,E2 -9820.488} C_VEL
LIN {X 0,Y 424.999,Z 521.306,A -85,B 0,C 180,E1 -9822.414,E2 -9822.414} C_VEL
LIN {X 0,Y 425.647,Z 512.655,A -85,B 0,C 180,E1 -9824.096,E2 -9824.096} C_VEL
LIN {X 0,Y 426.422,Z 502.235,A -85,B 0,C 180,E1 -9825.78,E2 -9825.78} C_VEL
LIN {X 0,Y 427.505,Z 490.566,A -85,B 0,C 180,E1 -9827.34,E2 -9827.34} C_VEL
LIN {X 0,Y 428.489,Z 478.804,A -85,B 0,C 180,E1 -9828.653,E2 -9828.653} C_VEL
LIN {X 0,Y 429.643,Z 465.957,A -85,B 0,C 180,E1 -9829.842,E2 -9829.842} C_VEL
LIN {X 0,Y 430.663,Z 453.581,A -85,B 0,C 180,E1 -9830.79,E2 -9830.79} C_VEL
LIN {X 0,Y 431.733,Z 439.786,A -85,B 0,C 180,E1 -9831.642,E2 -9831.642} C_VEL
LIN {X 0,Y 432.705,Z 424.363,A -85,B 0,C 180,E1 -9832.372,E2 -9832.372} C_VEL
LIN {X 0,Y 431.356,Z 409.359,A -85,B 0,C 180,E1 -9832.996,E2 -9832.996} C_VEL
LIN {X 0,Y 428.954,Z 393.434,A -85,B 0,C 180,E1 -9833.508,E2 -9833.508} C_VEL
LIN {X 0,Y 426.954,Z 383.369,A -85,B 0,C 180,E1 -9833.825,E2 -9833.825} C_VEL
LIN {X 0,Y 428.017,Z 369.563,A -85,B 0,C 180,E1 -9836.843,E2 -9836.843} C_VEL
LIN {X 0,Y 429.6,Z 355.814,A -85,B 0,C 180,E1 -9840.09,E2 -9840.09} C_VEL
LIN {X 0,Y 431.423,Z 344.329,A -85,B 0,C 180,E1 -9843.074,E2 -9843.074} C_VEL
LIN {X 0,Y 433.731,Z 334.671,A -85,B 0,C 180,E1 -9845.887,E2 -9845.887} C_VEL
LIN {X 0,Y 433.953,Z 333.521,A -85,B 0,C 180,E1 -9846.257,E2 -9846.257} C_VEL
LIN {X 0,Y 433.041,Z 328.976,A -85,B 0,C 180,E1 -9848.077,E2 -9848.077} C_VEL
LIN {X 0,Y 431.715,Z 323.804,A -85,B 0,C 180,E1 -9850.63,E2 -9850.63} C_VEL
LIN {X 0,Y 430.532,Z 319.754,A -85,B 0,C 180,E1 -9853.284,E2 -9853.284} C_VEL
LIN {X 0,Y 429.663,Z 316.843,A -85,B 0,C 180,E1 -9856.031,E2 -9856.031} C_VEL
LIN {X 0,Y 428.997,Z 315.051,A -85,B 0,C 180,E1 -9858.903,E2 -9858.903} C_VEL
LIN {X 0,Y 428.545,Z 314.271,A -85,B 0,C 180,E1 -9861.924,E2 -9861.924} C_VEL
LIN {X 0,Y 428.293,Z 314.287,A -85,B 0,C 180,E1 -9863.791,E2 -9863.791} C_VEL
LIN {X 0,Y 427.68,Z 314.987,A -85,B 0,C 180,E1 -9867.161,E2 -9867.161} C_VEL
LIN {X 0,Y 427.147,Z 316.385,A -85,B 0,C 180,E1 -9870.696,E2 -9870.696} C_VEL
LIN {X 0,Y 426.867,Z 317.869,A -85,B 0,C 180,E1 -9873.607,E2 -9873.607} C_VEL
LIN {X 0,Y 426.603,Z 319.72,A -85,B 0,C 180,E1 -9876.71,E2 -9876.71} C_VEL
LIN {X 0,Y 426.385,Z 321.894,A -85,B 0,C 180,E1 -9879.972,E2 -9879.972} C_VEL
LIN {X 0,Y 426.295,Z 323.265,A -85,B 0,C 180,E1 -9881.668,E2 -9881.668} C_VEL
LIN {X 0,Y 431.642,Z 336.031,A -85,B 0,C 180,E1 -9882.684,E2 -9882.684} C_VEL
LIN {X 0,Y 432.915,Z 340.182,A -85,B 0,C 180,E1 -9883.01,E2 -9883.01} C_VEL
LIN {X 0,Y 432.094,Z 353.249,A -85,B 0,C 180,E1 -9883.837,E2 -9883.837} C_VEL
LIN {X 0,Y 431.095,Z 366.162,A -85,B 0,C 180,E1 -9884.88,E2 -9884.88} C_VEL
LIN {X 0,Y 430.227,Z 376.585,A -85,B 0,C 180,E1 -9885.937,E2 -9885.937} C_VEL
LIN {X 0,Y 429.282,Z 387.091,A -85,B 0,C 180,E1 -9887.231,E2 -9887.231} C_VEL
LIN {X 0,Y 428.333,Z 396.406,A -85,B 0,C 180,E1 -9888.645,E2 -9888.645} C_VEL
LIN {X 0,Y 427.654,Z 403.905,A -85,B 0,C 180,E1 -9890.064,E2 -9890.064} C_VEL
LIN {X 0,Y 426.986,Z 410.003,A -85,B 0,C 180,E1 -9891.481,E2 -9891.481} C_VEL
LIN {X 0,Y 426.502,Z 414.87,A -85,B 0,C 180,E1 -9892.901,E2 -9892.901} C_VEL
LIN {X 0,Y 425.933,Z 418.689,A -85,B 0,C 180,E1 -9894.318,E2 -9894.318} C_VEL
LIN {X 0,Y 425.851,Z 420.636,A -85,B 0,C 180,E1 -9895.267,E2 -9895.267} C_VEL
LIN {X 0,Y 425.774,Z 422.145,A -85,B 0,C 180,E1 -9896.214,E2 -9896.214} C_VEL
LIN {X 0,Y 425.38,Z 423.976,A -85,B 0,C 180,E1 -9898.107,E2 -9898.107} C_VEL
LIN {X 0,Y 425.303,Z 424.295,A -85,B 0,C 180,E1 -9899.053,E2 -9899.053} C_VEL
LIN {X 0,Y 425.256,Z 424.211,A -85,B 0,C 180,E1 -9900,E2 -9900} C_VEL
LIN {X 0,Y 425.261,Z 423.699,A -85,B 0,C 180,E1 -9900.947,E2 -9900.947} C_VEL
LIN {X 0,Y 425.105,Z 421.548,A -85,B 0,C 180,E1 -9902.843,E2 -9902.843} C_VEL
LIN {X 0,Y 425.263,Z 418.799,A -85,B 0,C 180,E1 -9904.265,E2 -9904.265} C_VEL
LIN {X 0,Y 425.482,Z 415.06,A -85,B 0,C 180,E1 -9905.688,E2 -9905.688} C_VEL
LIN {X 0,Y 425.792,Z 410.244,A -85,B 0,C 180,E1 -9907.111,E2 -9907.111} C_VEL
LIN {X 0,Y 426.177,Z 403.102,A -85,B 0,C 180,E1 -9908.774,E2 -9908.774} C_VEL
LIN {X 0,Y 426.601,Z 395.404,A -85,B 0,C 180,E1 -9910.201,E2 -9910.201} C_VEL
LIN {X 0,Y 427.04,Z 385.976,A -85,B 0,C 180,E1 -9911.631,E2 -9911.631} C_VEL
LIN {X 0,Y 427.787,Z 375.256,A -85,B 0,C 180,E1 -9912.935,E2 -9912.935} C_VEL
LIN {X 0,Y 428.397,Z 363.233,A -85,B 0,C 180,E1 -9914.125,E2 -9914.125} C_VEL
LIN {X 0,Y 428.984,Z 350.758,A -85,B 0,C 180,E1 -9915.102,E2 -9915.102} C_VEL
LIN {X 0,Y 429.541,Z 337.668,A -85,B 0,C 180,E1 -9915.906,E2 -9915.906} C_VEL
LIN {X 0,Y 429.729,Z 332.952,A -85,B 0,C 180,E1 -9916.143,E2 -9916.143} C_VEL
LIN {X 0,Y 426.293,Z 319.844,A -85,B 0,C 180,E1 -9916.834,E2 -9916.834} C_VEL
LIN {X 0,Y 424.692,Z 313.635,A -85,B 0,C 180,E1 -9917.12,E2 -9917.12} C_VEL
LIN {X 0,Y 424.684,Z 310.067,A -85,B 0,C 180,E1 -9920.336,E2 -9920.336} C_VEL
LIN {X 0,Y 424.718,Z 306.74,A -85,B 0,C 180,E1 -9923.4,E2 -9923.4} C_VEL
LIN {X 0,Y 424.722,Z 303.236,A -85,B 0,C 180,E1 -9926.676,E2 -9926.676} C_VEL
LIN {X 0,Y 424.77,Z 299.964,A -85,B 0,C 180,E1 -9929.76,E2 -9929.76} C_VEL
LIN {X 0,Y 424.788,Z 298.832,A -85,B 0,C 180,E1 -9930.856,E2 -9930.856} C_VEL
LIN {X 0,Y 424.896,Z 298.186,A -85,B 0,C 180,E1 -9932.481,E2 -9932.481} C_VEL
LIN {X 0,Y 425.205,Z 298.147,A -85,B 0,C 180,E1 -9935.345,E2 -9935.345} C_VEL
LIN {X 0,Y 425.279,Z 298.135,A -85,B 0,C 180,E1 -9937.694,E2 -9937.694} C_VEL
LIN {X 0,Y 425.282,Z 298.133,A -85,B 0,C 180,E1 -9940.52,E2 -9940.52} C_VEL
LIN {X 0,Y 425.259,Z 298.133,A -85,B 0,C 180,E1 -9943.351,E2 -9943.351} C_VEL
LIN {X 0,Y 425.258,Z 298.139,A -85,B 0,C 180,E1 -9946.043,E2 -9946.043} C_VEL
LIN {X 0,Y 425.258,Z 298.188,A -85,B 0,C 180,E1 -9948.125,E2 -9948.125} C_VEL
LIN {X 0,Y 425.465,Z 300.637,A -85,B 0,C 180,E1 -9949.893,E2 -9949.893} C_VEL
LIN {X 0,Y 425.353,Z 305.596,A -85,B 0,C 180,E1 -9953.5,E2 -9953.5} C_VEL
LIN {X 0,Y 425.352,Z 308.703,A -85,B 0,C 180,E1 -9955.821,E2 -9955.821} C_VEL
LIN {X 0,Y 425.264,Z 313.381,A -85,B 0,C 180,E1 -9959.245,E2 -9959.245} C_VEL
LIN {X 0,Y 425.266,Z 316.353,A -85,B 0,C 180,E1 -9961.363,E2 -9961.363} C_VEL
LIN {X 0,Y 425.19,Z 321.105,A -85,B 0,C 180,E1 -9964.548,E2 -9964.548} C_VEL
LIN {X 0,Y 425.209,Z 323.461,A -85,B 0,C 180,E1 -9966.021,E2 -9966.021} C_VEL
LIN {X 0,Y 431.191,Z 339.749,A -85,B 0,C 180,E1 -9966.777,E2 -9966.777} C_VEL
LIN {X 0,Y 434.592,Z 350.554,A -85,B 0,C 180,E1 -9967.363,E2 -9967.363} C_VEL
LIN {X 0,Y 433.944,Z 364.527,A -85,B 0,C 180,E1 -9967.987,E2 -9967.987} C_VEL
LIN {X 0,Y 433.068,Z 378.977,A -85,B 0,C 180,E1 -9968.833,E2 -9968.833} C_VEL
LIN {X 0,Y 432.081,Z 391.871,A -85,B 0,C 180,E1 -9969.779,E2 -9969.779} C_VEL
LIN {X 0,Y 430.928,Z 405.036,A -85,B 0,C 180,E1 -9970.963,E2 -9970.963} C_VEL
LIN {X 0,Y 429.885,Z 415.955,A -85,B 0,C 180,E1 -9972.149,E2 -9972.149} C_VEL
LIN {X 0,Y 428.733,Z 427.009,A -85,B 0,C 180,E1 -9973.574,E2 -9973.574} C_VEL
LIN {X 0,Y 427.782,Z 436.298,A -85,B 0,C 180,E1 -9975.004,E2 -9975.004} C_VEL
LIN {X 0,Y 426.883,Z 445.405,A -85,B 0,C 180,E1 -9976.674,E2 -9976.674} C_VEL
LIN {X 0,Y 426.253,Z 451.996,A -85,B 0,C 180,E1 -9978.106,E2 -9978.106} C_VEL
LIN {X 0,Y 425.564,Z 459.233,A -85,B 0,C 180,E1 -9980.014,E2 -9980.014} C_VEL
LIN {X 0,Y 425.06,Z 464.967,A -85,B 0,C 180,E1 -9981.921,E2 -9981.921} C_VEL
LIN {X 0,Y 424.801,Z 468.35,A -85,B 0,C 180,E1 -9983.349,E2 -9983.349} C_VEL
LIN {X 0,Y 424.602,Z 470.637,A -85,B 0,C 180,E1 -9984.549,E2 -9984.549} C_VEL
LIN {X 0,Y 423.92,Z 471.979,A -85,B 0,C 180,E1 -9985.323,E2 -9985.323} C_VEL
LIN {X 0,Y 420.977,Z 473.841,A -85,B 0,C 180,E1 -9986.583,E2 -9986.583} C_VEL
LIN {X 0,Y 418.464,Z 474.977,A -85,B 0,C 180,E1 -9987.608,E2 -9987.608} C_VEL
LIN {X 0,Y 417.352,Z 475.55,A -85,B 0,C 180,E1 -9988.405,E2 -9988.405} C_VEL
LIN {X 0,Y 417.245,Z 475.675,A -85,B 0,C 180,E1 -9988.677,E2 -9988.677} C_VEL
LIN {X 0,Y 417.189,Z 475.996,A -85,B 0,C 180,E1 -9990,E2 -9990} C_VEL
LIN {X 0,Y 417.323,Z 475.436,A -85,B 0,C 180,E1 -9991.93,E2 -9991.93} C_VEL
LIN {X 0,Y 417.511,Z 473.777,A -85,B 0,C 180,E1 -9993.861,E2 -9993.861} C_VEL
LIN {X 0,Y 417.559,Z 471.004,A -85,B 0,C 180,E1 -9995.796,E2 -9995.796} C_VEL
LIN {X 0,Y 417.967,Z 467.005,A -85,B 0,C 180,E1 -9997.731,E2 -9997.731} C_VEL
LIN {X 0,Y 418.412,Z 461.698,A -85,B 0,C 180,E1 -9999.67,E2 -9999.67} C_VEL
LIN {X 0,Y 419.114,Z 454.919,A -85,B 0,C 180,E1 -10001.608,E2 -10001.608} C_VEL
LIN {X 0,Y 419.861,Z 447.656,A -85,B 0,C 180,E1 -10003.306,E2 -10003.306} C_VEL
LIN {X 0,Y 420.723,Z 438.892,A -85,B 0,C 180,E1 -10005.006,E2 -10005.006} C_VEL
LIN {X 0,Y 421.906,Z 428.273,A -85,B 0,C 180,E1 -10006.699,E2 -10006.699} C_VEL
LIN {X 0,Y 423.039,Z 417.357,A -85,B 0,C 180,E1 -10008.149,E2 -10008.149} C_VEL
LIN {X 0,Y 424.278,Z 405.354,A -85,B 0,C 180,E1 -10009.473,E2 -10009.473} C_VEL
LIN {X 0,Y 425.489,Z 392.097,A -85,B 0,C 180,E1 -10010.674,E2 -10010.674} C_VEL
LIN {X 0,Y 426.574,Z 379.123,A -85,B 0,C 180,E1 -10011.631,E2 -10011.631} C_VEL
LIN {X 0,Y 427.449,Z 365.255,A -85,B 0,C 180,E1 -10012.453,E2 -10012.453} C_VEL
LIN {X 0,Y 427.966,Z 351.81,A -85,B 0,C 180,E1 -10013.074,E2 -10013.074} C_VEL
LIN {X 0,Y 423.137,Z 337.083,A -85,B 0,C 180,E1 -10013.891,E2 -10013.891} C_VEL
LIN {X 0,Y 418.223,Z 324.01,A -85,B 0,C 180,E1 -10014.523,E2 -10014.523} C_VEL
LIN {X 0,Y 418.249,Z 320.031,A -85,B 0,C 180,E1 -10017.053,E2 -10017.053} C_VEL
LIN {X 0,Y 418.294,Z 316.969,A -85,B 0,C 180,E1 -10019.16,E2 -10019.16} C_VEL
LIN {X 0,Y 418.3,Z 311.846,A -85,B 0,C 180,E1 -10022.853,E2 -10022.853} C_VEL
LIN {X 0,Y 418.341,Z 307.278,A -85,B 0,C 180,E1 -10026.256,E2 -10026.256} C_VEL
LIN {X 0,Y 418.442,Z 302.951,A -85,B 0,C 180,E1 -10029.412,E2 -10029.412} C_VEL
LIN {X 0,Y 418.423,Z 300.882,A -85,B 0,C 180,E1 -10030.924,E2 -10030.924} C_VEL
LIN {X 0,Y 418.204,Z 299.021,A -85,B 0,C 180,E1 -10032.317,E2 -10032.317} C_VEL
LIN {X 0,Y 418.236,Z 299.017,A -85,B 0,C 180,E1 -10035.108,E2 -10035.108} C_VEL
LIN {X 0,Y 418.241,Z 299.014,A -85,B 0,C 180,E1 -10037.767,E2 -10037.767} C_VEL
LIN {X 0,Y 418.242,Z 299.009,A -85,B 0,C 180,E1 -10040.621,E2 -10040.621} C_VEL
LIN {X 0,Y 418.243,Z 299.011,A -85,B 0,C 180,E1 -10043.976,E2 -10043.976} C_VEL
LIN {X 0,Y 418.258,Z 299.008,A -85,B 0,C 180,E1 -10047.156,E2 -10047.156} C_VEL
LIN {X 0,Y 418.258,Z 299.009,A -85,B 0,C 180,E1 -10050.837,E2 -10050.837} C_VEL
LIN {X 0,Y 418.228,Z 299.006,A -85,B 0,C 180,E1 -10054.093,E2 -10054.093} C_VEL
LIN {X 0,Y 418.237,Z 299.007,A -85,B 0,C 180,E1 -10057.264,E2 -10057.264} C_VEL
LIN {X 0,Y 418.283,Z 299.01,A -85,B 0,C 180,E1 -10060.364,E2 -10060.364} C_VEL
LIN {X 0,Y 418.316,Z 298.992,A -85,B 0,C 180,E1 -10063.404,E2 -10063.404} C_VEL
LIN {X 0,Y 418.347,Z 298.994,A -85,B 0,C 180,E1 -10066.999,E2 -10066.999} C_VEL
LIN {X 0,Y 418.338,Z 299,A -85,B 0,C 180,E1 -10070.328,E2 -10070.328} C_VEL
LIN {X 0,Y 418.443,Z 298.978,A -85,B 0,C 180,E1 -10073.248,E2 -10073.248} C_VEL
LIN {X 0,Y 418.328,Z 298.994,A -85,B 0,C 180,E1 -10075.181,E2 -10075.181} C_VEL
LIN {X 0,Y 418.543,Z 298.973,A -85,B 0,C 180,E1 -10078.075,E2 -10078.075} C_VEL
LIN {X 0,Y 418.672,Z 298.945,A -85,B 0,C 180,E1 -10080,E2 -10080} C_VEL
LIN {X 0,Y 418.488,Z 298.98,A -85,B 0,C 180,E1 -10082.888,E2 -10082.888} C_VEL
LIN {X 0,Y 418.495,Z 298.969,A -85,B 0,C 180,E1 -10085.783,E2 -10085.783} C_VEL
LIN {X 0,Y 418.378,Z 298.995,A -85,B 0,C 180,E1 -10088.695,E2 -10088.695} C_VEL
LIN {X 0,Y 418.316,Z 298.99,A -85,B 0,C 180,E1 -10091.631,E2 -10091.631} C_VEL
LIN {X 0,Y 418.299,Z 299.004,A -85,B 0,C 180,E1 -10094.597,E2 -10094.597} C_VEL
LIN {X 0,Y 418.279,Z 299.003,A -85,B 0,C 180,E1 -10097.604,E2 -10097.604} C_VEL
LIN {X 0,Y 418.25,Z 299.004,A -85,B 0,C 180,E1 -10100.663,E2 -10100.663} C_VEL
LIN {X 0,Y 418.272,Z 299.011,A -85,B 0,C 180,E1 -10103.782,E2 -10103.782} C_VEL
LIN {X 0,Y 418.223,Z 299.006,A -85,B 0,C 180,E1 -10107.047,E2 -10107.047} C_VEL
LIN {X 0,Y 418.241,Z 299.015,A -85,B 0,C 180,E1 -10110.272,E2 -10110.272} C_VEL
LIN {X 0,Y 418.248,Z 299.013,A -85,B 0,C 180,E1 -10113.677,E2 -10113.677} C_VEL
LIN {X 0,Y 418.237,Z 299.014,A -85,B 0,C 180,E1 -10117.224,E2 -10117.224} C_VEL
LIN {X 0,Y 418.242,Z 299.013,A -85,B 0,C 180,E1 -10119.683,E2 -10119.683} C_VEL
LIN {X 0,Y 418.229,Z 299.009,A -85,B 0,C 180,E1 -10122.321,E2 -10122.321} C_VEL
LIN {X 0,Y 418.25,Z 299.204,A -85,B 0,C 180,E1 -10124.032,E2 -10124.032} C_VEL
LIN {X 0,Y 420.816,Z 309.486,A -85,B 0,C 180,E1 -10127.294,E2 -10127.294} C_VEL
LIN {X 0,Y 423.405,Z 319.961,A -85,B 0,C 180,E1 -10130.399,E2 -10130.399} C_VEL
LIN {X 0,Y 426.179,Z 331.429,A -85,B 0,C 180,E1 -10133.583,E2 -10133.583} C_VEL
LIN {X 0,Y 424.724,Z 343.006,A -85,B 0,C 180,E1 -10136.335,E2 -10136.335} C_VEL
LIN {X 0,Y 422.832,Z 358.046,A -85,B 0,C 180,E1 -10139.803,E2 -10139.803} C_VEL
LIN {X 0,Y 421.371,Z 372.111,A -85,B 0,C 180,E1 -10142.967,E2 -10142.967} C_VEL
LIN {X 0,Y 420.283,Z 385.062,A -85,B 0,C 180,E1 -10145.815,E2 -10145.815} C_VEL
LIN {X 0,Y 424.08,Z 406.626,A -85,B 0,C 180,E1 -10146.52,E2 -10146.52} C_VEL
LIN {X 0,Y 425.774,Z 422.012,A -85,B 0,C 180,E1 -10147.165,E2 -10147.165} C_VEL
LIN {X 0,Y 425.972,Z 425.732,A -85,B 0,C 180,E1 -10147.336,E2 -10147.336} C_VEL
LIN {X 0,Y 424.96,Z 440.863,A -85,B 0,C 180,E1 -10148.093,E2 -10148.093} C_VEL
LIN {X 0,Y 423.81,Z 454.736,A -85,B 0,C 180,E1 -10148.986,E2 -10148.986} C_VEL
LIN {X 0,Y 422.564,Z 468.216,A -85,B 0,C 180,E1 -10150.065,E2 -10150.065} C_VEL
LIN {X 0,Y 421.47,Z 480.599,A -85,B 0,C 180,E1 -10151.277,E2 -10151.277} C_VEL
LIN {X 0,Y 420.29,Z 492.934,A -85,B 0,C 180,E1 -10152.734,E2 -10152.734} C_VEL
LIN {X 0,Y 419.391,Z 503.299,A -85,B 0,C 180,E1 -10154.198,E2 -10154.198} C_VEL
LIN {X 0,Y 418.537,Z 513.427,A -85,B 0,C 180,E1 -10155.908,E2 -10155.908} C_VEL
LIN {X 0,Y 417.898,Z 522.919,A -85,B 0,C 180,E1 -10157.865,E2 -10157.865} C_VEL
LIN {X 0,Y 417.512,Z 530.598,A -85,B 0,C 180,E1 -10159.82,E2 -10159.82} C_VEL
LIN {X 0,Y 417.37,Z 536.707,A -85,B 0,C 180,E1 -10161.771,E2 -10161.771} C_VEL
LIN {X 0,Y 417.379,Z 540.805,A -85,B 0,C 180,E1 -10163.445,E2 -10163.445} C_VEL
LIN {X 0,Y 417.302,Z 543.984,A -85,B 0,C 180,E1 -10165.17,E2 -10165.17} C_VEL
LIN {X 0,Y 417.421,Z 546.411,A -85,B 0,C 180,E1 -10167.105,E2 -10167.105} C_VEL
LIN {X 0,Y 417.338,Z 547.619,A -85,B 0,C 180,E1 -10169.035,E2 -10169.035} C_VEL
LIN {X 0,Y 417.338,Z 547.619,A -85,B 0,C 180,E1 -10170.965,E2 -10170.965} C_VEL
LIN {X 0,Y 417.43,Z 546.414,A -85,B 0,C 180,E1 -10172.895,E2 -10172.895} C_VEL
LIN {X 0,Y 417.364,Z 543.99,A -85,B 0,C 180,E1 -10174.83,E2 -10174.83} C_VEL
LIN {X 0,Y 417.408,Z 540.316,A -85,B 0,C 180,E1 -10176.769,E2 -10176.769} C_VEL
LIN {X 0,Y 417.404,Z 535.294,A -85,B 0,C 180,E1 -10178.716,E2 -10178.716} C_VEL
LIN {X 0,Y 417.662,Z 528.823,A -85,B 0,C 180,E1 -10180.667,E2 -10180.667} C_VEL
LIN {X 0,Y 417.988,Z 520.69,A -85,B 0,C 180,E1 -10182.626,E2 -10182.626} C_VEL
LIN {X 0,Y 418.65,Z 512.037,A -85,B 0,C 180,E1 -10184.337,E2 -10184.337} C_VEL
LIN {X 0,Y 419.516,Z 501.621,A -85,B 0,C 180,E1 -10186.047,E2 -10186.047} C_VEL
LIN {X 0,Y 420.669,Z 489.851,A -85,B 0,C 180,E1 -10187.644,E2 -10187.644} C_VEL
LIN {X 0,Y 421.678,Z 478.193,A -85,B 0,C 180,E1 -10188.966,E2 -10188.966} C_VEL
LIN {X 0,Y 422.874,Z 465.349,A -85,B 0,C 180,E1 -10190.173,E2 -10190.173} C_VEL
LIN {X 0,Y 423.987,Z 452.982,A -85,B 0,C 180,E1 -10191.133,E2 -10191.133} C_VEL
LIN {X 0,Y 425.113,Z 439.062,A -85,B 0,C 180,E1 -10192.004,E2 -10192.004} C_VEL
LIN {X 0,Y 426.031,Z 424.091,A -85,B 0,C 180,E1 -10192.729,E2 -10192.729} C_VEL
LIN {X 0,Y 424.814,Z 410.87,A -85,B 0,C 180,E1 -10193.305,E2 -10193.305} C_VEL
LIN {X 0,Y 422.587,Z 395.336,A -85,B 0,C 180,E1 -10193.837,E2 -10193.837} C_VEL
LIN {X 0,Y 420.055,Z 382.728,A -85,B 0,C 180,E1 -10194.246,E2 -10194.246} C_VEL
LIN {X 0,Y 421.095,Z 370.309,A -85,B 0,C 180,E1 -10197.052,E2 -10197.052} C_VEL
LIN {X 0,Y 422.675,Z 357.464,A -85,B 0,C 180,E1 -10200.16,E2 -10200.16} C_VEL
LIN {X 0,Y 424.528,Z 346.35,A -85,B 0,C 180,E1 -10203.115,E2 -10203.115} C_VEL
LIN {X 0,Y 426.688,Z 337.422,A -85,B 0,C 180,E1 -10205.756,E2 -10205.756} C_VEL
LIN {X 0,Y 427.155,Z 335.642,A -85,B 0,C 180,E1 -10206.321,E2 -10206.321} C_VEL
LIN {X 0,Y 426.278,Z 331.089,A -85,B 0,C 180,E1 -10208.191,E2 -10208.191} C_VEL
LIN {X 0,Y 425.105,Z 326.461,A -85,B 0,C 180,E1 -10210.493,E2 -10210.493} C_VEL
LIN {X 0,Y 423.92,Z 322.308,A -85,B 0,C 180,E1 -10213.159,E2 -10213.159} C_VEL
LIN {X 0,Y 423.039,Z 319.445,A -85,B 0,C 180,E1 -10215.753,E2 -10215.753} C_VEL
LIN {X 0,Y 422.353,Z 317.534,A -85,B 0,C 180,E1 -10218.487,E2 -10218.487} C_VEL
LIN {X 0,Y 421.827,Z 316.5,A -85,B 0,C 180,E1 -10221.542,E2 -10221.542} C_VEL
LIN {X 0,Y 421.372,Z 316.401,A -85,B 0,C 180,E1 -10224.285,E2 -10224.285} C_VEL
LIN {X 0,Y 420.717,Z 317.09,A -85,B 0,C 180,E1 -10227.686,E2 -10227.686} C_VEL
LIN {X 0,Y 420.249,Z 318.342,A -85,B 0,C 180,E1 -10230.989,E2 -10230.989} C_VEL
LIN {X 0,Y 419.911,Z 319.929,A -85,B 0,C 180,E1 -10234.205,E2 -10234.205} C_VEL
LIN {X 0,Y 419.678,Z 321.754,A -85,B 0,C 180,E1 -10237.346,E2 -10237.346} C_VEL
LIN {X 0,Y 419.376,Z 324.16,A -85,B 0,C 180,E1 -10240.926,E2 -10240.926} C_VEL
LIN {X 0,Y 419.377,Z 324.333,A -85,B 0,C 180,E1 -10241.148,E2 -10241.148} C_VEL
LIN {X 0,Y 421.776,Z 329.77,A -85,B 0,C 180,E1 -10241.601,E2 -10241.601} C_VEL
LIN {X 0,Y 426.259,Z 340.985,A -85,B 0,C 180,E1 -10242.565,E2 -10242.565} C_VEL
LIN {X 0,Y 426.523,Z 342.094,A -85,B 0,C 180,E1 -10242.652,E2 -10242.652} C_VEL
LIN {X 0,Y 425.587,Z 355.519,A -85,B 0,C 180,E1 -10243.548,E2 -10243.548} C_VEL
LIN {X 0,Y 424.596,Z 367.394,A -85,B 0,C 180,E1 -10244.535,E2 -10244.535} C_VEL
LIN {X 0,Y 423.58,Z 378.695,A -85,B 0,C 180,E1 -10245.712,E2 -10245.712} C_VEL
LIN {X 0,Y 422.577,Z 388.961,A -85,B 0,C 180,E1 -10247.025,E2 -10247.025} C_VEL
LIN {X 0,Y 421.569,Z 398.038,A -85,B 0,C 180,E1 -10248.46,E2 -10248.46} C_VEL
LIN {X 0,Y 420.834,Z 405.455,A -85,B 0,C 180,E1 -10249.901,E2 -10249.901} C_VEL
LIN {X 0,Y 420.12,Z 411.48,A -85,B 0,C 180,E1 -10251.341,E2 -10251.341} C_VEL
LIN {X 0,Y 419.598,Z 416.266,A -85,B 0,C 180,E1 -10252.784,E2 -10252.784} C_VEL
LIN {X 0,Y 418.99,Z 419.995,A -85,B 0,C 180,E1 -10254.224,E2 -10254.224} C_VEL
LIN {X 0,Y 418.903,Z 421.89,A -85,B 0,C 180,E1 -10255.188,E2 -10255.188} C_VEL
LIN {X 0,Y 418.791,Z 423.352,A -85,B 0,C 180,E1 -10256.151,E2 -10256.151} C_VEL
LIN {X 0,Y 418.378,Z 425.119,A -85,B 0,C 180,E1 -10258.075,E2 -10258.075} C_VEL
LIN {X 0,Y 418.293,Z 425.409,A -85,B 0,C 180,E1 -10259.037,E2 -10259.037} C_VEL
LIN {X 0,Y 418.238,Z 425.278,A -85,B 0,C 180,E1 -10260,E2 -10260} C_VEL
LIN {X 0,Y 418.24,Z 424.735,A -85,B 0,C 180,E1 -10260.963,E2 -10260.963} C_VEL
LIN {X 0,Y 418.13,Z 423.821,A -85,B 0,C 180,E1 -10261.927,E2 -10261.927} C_VEL
LIN {X 0,Y 418.079,Z 422.505,A -85,B 0,C 180,E1 -10262.891,E2 -10262.891} C_VEL
LIN {X 0,Y 418.248,Z 419.694,A -85,B 0,C 180,E1 -10264.337,E2 -10264.337} C_VEL
LIN {X 0,Y 418.486,Z 415.892,A -85,B 0,C 180,E1 -10265.783,E2 -10265.783} C_VEL
LIN {X 0,Y 418.802,Z 411.011,A -85,B 0,C 180,E1 -10267.23,E2 -10267.23} C_VEL
LIN {X 0,Y 419.195,Z 403.775,A -85,B 0,C 180,E1 -10268.922,E2 -10268.922} C_VEL
LIN {X 0,Y 419.652,Z 396.008,A -85,B 0,C 180,E1 -10270.372,E2 -10270.372} C_VEL
LIN {X 0,Y 420.127,Z 386.514,A -85,B 0,C 180,E1 -10271.825,E2 -10271.825} C_VEL
LIN {X 0,Y 420.889,Z 375.694,A -85,B 0,C 180,E1 -10273.151,E2 -10273.151} C_VEL
LIN {X 0,Y 421.468,Z 364.895,A -85,B 0,C 180,E1 -10274.239,E2 -10274.239} C_VEL
LIN {X 0,Y 422.058,Z 352.508,A -85,B 0,C 180,E1 -10275.248,E2 -10275.248} C_VEL
LIN {X 0,Y 422.673,Z 338.878,A -85,B 0,C 180,E1 -10276.109,E2 -10276.109} C_VEL
LIN {X 0,Y 422.877,Z 334.245,A -85,B 0,C 180,E1 -10276.349,E2 -10276.349} C_VEL
LIN {X 0,Y 419.399,Z 320.981,A -85,B 0,C 180,E1 -10277.074,E2 -10277.074} C_VEL
LIN {X 0,Y 417.66,Z 314.2,A -85,B 0,C 180,E1 -10277.366,E2 -10277.366} C_VEL
LIN {X 0,Y 417.638,Z 310.509,A -85,B 0,C 180,E1 -10280.695,E2 -10280.695} C_VEL
LIN {X 0,Y 417.651,Z 307.124,A -85,B 0,C 180,E1 -10283.82,E2 -10283.82} C_VEL
LIN {X 0,Y 417.676,Z 303.704,A -85,B 0,C 180,E1 -10287.021,E2 -10287.021} C_VEL
LIN {X 0,Y 417.721,Z 300.23,A -85,B 0,C 180,E1 -10290.314,E2 -10290.314} C_VEL
LIN {X 0,Y 417.738,Z 299.085,A -85,B 0,C 180,E1 -10291.436,E2 -10291.436} C_VEL
LIN {X 0,Y 418.116,Z 299.028,A -85,B 0,C 180,E1 -10294.855,E2 -10294.855} C_VEL
LIN {X 0,Y 418.228,Z 299.013,A -85,B 0,C 180,E1 -10297.833,E2 -10297.833} C_VEL
LIN {X 0,Y 418.225,Z 299.012,A -85,B 0,C 180,E1 -10300.948,E2 -10300.948} C_VEL
LIN {X 0,Y 418.212,Z 299.011,A -85,B 0,C 180,E1 -10303.729,E2 -10303.729} C_VEL
LIN {X 0,Y 418.2,Z 299.019,A -85,B 0,C 180,E1 -10306.447,E2 -10306.447} C_VEL
LIN {X 0,Y 418.236,Z 299.13,A -85,B 0,C 180,E1 -10307.928,E2 -10307.928} C_VEL
LIN {X 0,Y 418.448,Z 302.436,A -85,B 0,C 180,E1 -10310.34,E2 -10310.34} C_VEL
LIN {X 0,Y 418.364,Z 307.075,A -85,B 0,C 180,E1 -10313.74,E2 -10313.74} C_VEL
LIN {X 0,Y 418.3,Z 311.668,A -85,B 0,C 180,E1 -10317.147,E2 -10317.147} C_VEL
LIN {X 0,Y 418.247,Z 315.224,A -85,B 0,C 180,E1 -10319.728,E2 -10319.728} C_VEL
LIN {X 0,Y 418.214,Z 320.005,A -85,B 0,C 180,E1 -10323.017,E2 -10323.017} C_VEL
LIN {X 0,Y 418.23,Z 324.017,A -85,B 0,C 180,E1 -10325.583,E2 -10325.583} C_VEL
LIN {X 0,Y 424.445,Z 340.942,A -85,B 0,C 180,E1 -10326.405,E2 -10326.405} C_VEL
LIN {X 0,Y 427.977,Z 352.074,A -85,B 0,C 180,E1 -10327.034,E2 -10327.034} C_VEL
LIN {X 0,Y 427.374,Z 365.688,A -85,B 0,C 180,E1 -10327.664,E2 -10327.664} C_VEL
LIN {X 0,Y 426.495,Z 379.57,A -85,B 0,C 180,E1 -10328.491,E2 -10328.491} C_VEL
LIN {X 0,Y 425.466,Z 392.468,A -85,B 0,C 180,E1 -10329.45,E2 -10329.45} C_VEL
LIN {X 0,Y 424.239,Z 405.638,A -85,B 0,C 180,E1 -10330.651,E2 -10330.651} C_VEL
LIN {X 0,Y 423.156,Z 416.558,A -85,B 0,C 180,E1 -10331.856,E2 -10331.856} C_VEL
LIN {X 0,Y 421.962,Z 427.614,A -85,B 0,C 180,E1 -10333.303,E2 -10333.303} C_VEL
LIN {X 0,Y 420.946,Z 436.905,A -85,B 0,C 180,E1 -10334.754,E2 -10334.754} C_VEL
LIN {X 0,Y 419.982,Z 446.014,A -85,B 0,C 180,E1 -10336.451,E2 -10336.451} C_VEL
LIN {X 0,Y 419.314,Z 452.605,A -85,B 0,C 180,E1 -10337.906,E2 -10337.906} C_VEL
LIN {X 0,Y 418.582,Z 459.842,A -85,B 0,C 180,E1 -10339.846,E2 -10339.846} C_VEL
LIN {X 0,Y 418.052,Z 465.576,A -85,B 0,C 180,E1 -10341.784,E2 -10341.784} C_VEL
LIN {X 0,Y 417.761,Z 468.96,A -85,B 0,C 180,E1 -10343.237,E2 -10343.237} C_VEL
LIN {X 0,Y 417.588,Z 472.399,A -85,B 0,C 180,E1 -10345.173,E2 -10345.173} C_VEL
LIN {X 0,Y 417.489,Z 474.668,A -85,B 0,C 180,E1 -10347.105,E2 -10347.105} C_VEL
LIN {X 0,Y 417.245,Z 475.675,A -85,B 0,C 180,E1 -10348.677,E2 -10348.677} C_VEL
LIN {X 0,Y 416.529,Z 475.994,A -85,B 0,C 180,E1 -10349.481,E2 -10349.481} C_VEL
LIN {X 0,Y 413.673,Z 476.189,A -85,B 0,C 180,E1 -10350.79,E2 -10350.79} C_VEL
LIN {X 0,Y 411.357,Z 476.001,A -85,B 0,C 180,E1 -10351.847,E2 -10351.847} C_VEL
LIN {X 0,Y 410.462,Z 475.563,A -85,B 0,C 180,E1 -10352.662,E2 -10352.662} C_VEL
LIN {X 0,Y 410.44,Z 475.351,A -85,B 0,C 180,E1 -10352.936,E2 -10352.936} C_VEL
LIN {X 0,Y 410.546,Z 473.137,A -85,B 0,C 180,E1 -10354.91,E2 -10354.91} C_VEL
LIN {X 0,Y 410.759,Z 469.765,A -85,B 0,C 180,E1 -10356.879,E2 -10356.879} C_VEL
LIN {X 0,Y 411.15,Z 465.133,A -85,B 0,C 180,E1 -10358.849,E2 -10358.849} C_VEL
LIN {X 0,Y 411.755,Z 459.111,A -85,B 0,C 180,E1 -10360.821,E2 -10360.821} C_VEL
LIN {X 0,Y 412.586,Z 451.525,A -85,B 0,C 180,E1 -10362.794,E2 -10362.794} C_VEL
LIN {X 0,Y 413.422,Z 443.642,A -85,B 0,C 180,E1 -10364.481,E2 -10364.481} C_VEL
LIN {X 0,Y 414.419,Z 435.181,A -85,B 0,C 180,E1 -10365.996,E2 -10365.996} C_VEL
LIN {X 0,Y 415.564,Z 425.415,A -85,B 0,C 180,E1 -10367.469,E2 -10367.469} C_VEL
LIN {X 0,Y 416.677,Z 414.423,A -85,B 0,C 180,E1 -10368.871,E2 -10368.871} C_VEL
LIN {X 0,Y 418.007,Z 402.192,A -85,B 0,C 180,E1 -10370.161,E2 -10370.161} C_VEL
LIN {X 0,Y 419.144,Z 389.624,A -85,B 0,C 180,E1 -10371.26,E2 -10371.26} C_VEL
LIN {X 0,Y 420.234,Z 375.891,A -85,B 0,C 180,E1 -10372.233,E2 -10372.233} C_VEL
LIN {X 0,Y 421.128,Z 361.315,A -85,B 0,C 180,E1 -10373.047,E2 -10373.047} C_VEL
LIN {X 0,Y 421.344,Z 353.449,A -85,B 0,C 180,E1 -10373.41,E2 -10373.41} C_VEL
LIN {X 0,Y 417.014,Z 339.914,A -85,B 0,C 180,E1 -10374.191,E2 -10374.191} C_VEL
LIN {X 0,Y 411.232,Z 324.581,A -85,B 0,C 180,E1 -10374.967,E2 -10374.967} C_VEL
LIN {X 0,Y 411.26,Z 319.019,A -85,B 0,C 180,E1 -10378.587,E2 -10378.587} C_VEL
LIN {X 0,Y 411.274,Z 314.207,A -85,B 0,C 180,E1 -10381.988,E2 -10381.988} C_VEL
LIN {X 0,Y 411.316,Z 309.44,A -85,B 0,C 180,E1 -10385.517,E2 -10385.517} C_VEL
LIN {X 0,Y 411.418,Z 305.83,A -85,B 0,C 180,E1 -10388.206,E2 -10388.206} C_VEL
LIN {X 0,Y 411.422,Z 302.706,A -85,B 0,C 180,E1 -10390.475,E2 -10390.475} C_VEL
LIN {X 0,Y 411.164,Z 299.897,A -85,B 0,C 180,E1 -10392.693,E2 -10392.693} C_VEL
LIN {X 0,Y 411.168,Z 299.897,A -85,B 0,C 180,E1 -10395.881,E2 -10395.881} C_VEL
LIN {X 0,Y 411.164,Z 299.893,A -85,B 0,C 180,E1 -10398.772,E2 -10398.772} C_VEL
LIN {X 0,Y 411.19,Z 299.894,A -85,B 0,C 180,E1 -10402.026,E2 -10402.026} C_VEL
LIN {X 0,Y 411.206,Z 299.887,A -85,B 0,C 180,E1 -10405.666,E2 -10405.666} C_VEL
LIN {X 0,Y 411.188,Z 299.887,A -85,B 0,C 180,E1 -10409.152,E2 -10409.152} C_VEL
LIN {X 0,Y 411.175,Z 299.891,A -85,B 0,C 180,E1 -10411.407,E2 -10411.407} C_VEL
LIN {X 0,Y 411.226,Z 299.881,A -85,B 0,C 180,E1 -10414.929,E2 -10414.929} C_VEL
LIN {X 0,Y 411.205,Z 299.88,A -85,B 0,C 180,E1 -10417.913,E2 -10417.913} C_VEL
LIN {X 0,Y 411.218,Z 299.886,A -85,B 0,C 180,E1 -10421.051,E2 -10421.051} C_VEL
LIN {X 0,Y 411.255,Z 299.878,A -85,B 0,C 180,E1 -10424.132,E2 -10424.132} C_VEL
LIN {X 0,Y 411.304,Z 299.87,A -85,B 0,C 180,E1 -10427.166,E2 -10427.166} C_VEL
LIN {X 0,Y 411.291,Z 299.875,A -85,B 0,C 180,E1 -10430.161,E2 -10430.161} C_VEL
LIN {X 0,Y 411.392,Z 299.857,A -85,B 0,C 180,E1 -10433.132,E2 -10433.132} C_VEL
LIN {X 0,Y 411.299,Z 299.868,A -85,B 0,C 180,E1 -10435.099,E2 -10435.099} C_VEL
LIN {X 0,Y 411.512,Z 299.848,A -85,B 0,C 180,E1 -10438.042,E2 -10438.042} C_VEL
LIN {X 0,Y 411.641,Z 299.82,A -85,B 0,C 180,E1 -10440,E2 -10440} C_VEL
LIN {X 0,Y 411.445,Z 299.858,A -85,B 0,C 180,E1 -10442.937,E2 -10442.937} C_VEL
LIN {X 0,Y 411.431,Z 299.855,A -85,B 0,C 180,E1 -10446.867,E2 -10446.867} C_VEL
LIN {X 0,Y 411.292,Z 299.872,A -85,B 0,C 180,E1 -10449.839,E2 -10449.839} C_VEL
LIN {X 0,Y 411.306,Z 299.874,A -85,B 0,C 180,E1 -10453.104,E2 -10453.104} C_VEL
LIN {X 0,Y 411.257,Z 299.871,A -85,B 0,C 180,E1 -10456.889,E2 -10456.889} C_VEL
LIN {X 0,Y 411.23,Z 299.886,A -85,B 0,C 180,E1 -10459.987,E2 -10459.987} C_VEL
LIN {X 0,Y 411.194,Z 299.886,A -85,B 0,C 180,E1 -10463.148,E2 -10463.148} C_VEL
LIN {X 0,Y 411.185,Z 299.881,A -85,B 0,C 180,E1 -10466.384,E2 -10466.384} C_VEL
LIN {X 0,Y 411.197,Z 299.889,A -85,B 0,C 180,E1 -10469.713,E2 -10469.713} C_VEL
LIN {X 0,Y 411.206,Z 299.889,A -85,B 0,C 180,E1 -10473.156,E2 -10473.156} C_VEL
LIN {X 0,Y 411.191,Z 299.892,A -85,B 0,C 180,E1 -10476.552,E2 -10476.552} C_VEL
LIN {X 0,Y 411.206,Z 299.889,A -85,B 0,C 180,E1 -10479.727,E2 -10479.727} C_VEL
LIN {X 0,Y 411.173,Z 299.886,A -85,B 0,C 180,E1 -10483.419,E2 -10483.419} C_VEL
LIN {X 0,Y 413.564,Z 309.605,A -85,B 0,C 180,E1 -10486.592,E2 -10486.592} C_VEL
LIN {X 0,Y 416.297,Z 320.6,A -85,B 0,C 180,E1 -10489.937,E2 -10489.937} C_VEL
LIN {X 0,Y 419.143,Z 332.309,A -85,B 0,C 180,E1 -10493.279,E2 -10493.279} C_VEL
LIN {X 0,Y 419.261,Z 333.915,A -85,B 0,C 180,E1 -10493.697,E2 -10493.697} C_VEL
LIN {X 0,Y 417.26,Z 348.061,A -85,B 0,C 180,E1 -10497.099,E2 -10497.099} C_VEL
LIN {X 0,Y 415.434,Z 363.094,A -85,B 0,C 180,E1 -10500.62,E2 -10500.62} C_VEL
LIN {X 0,Y 413.853,Z 378.623,A -85,B 0,C 180,E1 -10504.163,E2 -10504.163} C_VEL
LIN {X 0,Y 413.326,Z 384.093,A -85,B 0,C 180,E1 -10505.381,E2 -10505.381} C_VEL
LIN {X 0,Y 417.168,Z 405.45,A -85,B 0,C 180,E1 -10506.09,E2 -10506.09} C_VEL
LIN {X 0,Y 418.642,Z 417.933,A -85,B 0,C 180,E1 -10506.604,E2 -10506.604} C_VEL
LIN {X 0,Y 419.272,Z 427.464,A -85,B 0,C 180,E1 -10507.068,E2 -10507.068} C_VEL
LIN {X 0,Y 418.276,Z 441.118,A -85,B 0,C 180,E1 -10507.779,E2 -10507.779} C_VEL
LIN {X 0,Y 416.978,Z 455.734,A -85,B 0,C 180,E1 -10508.754,E2 -10508.754} C_VEL
LIN {X 0,Y 415.685,Z 468.918,A -85,B 0,C 180,E1 -10509.85,E2 -10509.85} C_VEL
LIN {X 0,Y 414.546,Z 481.079,A -85,B 0,C 180,E1 -10511.081,E2 -10511.081} C_VEL
LIN {X 0,Y 413.431,Z 492.325,A -85,B 0,C 180,E1 -10512.438,E2 -10512.438} C_VEL
LIN {X 0,Y 412.458,Z 502.687,A -85,B 0,C 180,E1 -10513.926,E2 -10513.926} C_VEL
LIN {X 0,Y 411.562,Z 512.814,A -85,B 0,C 180,E1 -10515.664,E2 -10515.664} C_VEL
LIN {X 0,Y 410.82,Z 522.3,A -85,B 0,C 180,E1 -10517.653,E2 -10517.653} C_VEL
LIN {X 0,Y 410.477,Z 529.986,A -85,B 0,C 180,E1 -10519.643,E2 -10519.643} C_VEL
LIN {X 0,Y 410.29,Z 536.093,A -85,B 0,C 180,E1 -10521.628,E2 -10521.628} C_VEL
LIN {X 0,Y 410.303,Z 540.453,A -85,B 0,C 180,E1 -10523.449,E2 -10523.449} C_VEL
LIN {X 0,Y 410.228,Z 543.375,A -85,B 0,C 180,E1 -10525.086,E2 -10525.086} C_VEL
LIN {X 0,Y 410.345,Z 545.802,A -85,B 0,C 180,E1 -10527.055,E2 -10527.055} C_VEL
LIN {X 0,Y 410.277,Z 547.011,A -85,B 0,C 180,E1 -10529.019,E2 -10529.019} C_VEL
LIN {X 0,Y 410.276,Z 547.012,A -85,B 0,C 180,E1 -10530.982,E2 -10530.982} C_VEL
LIN {X 0,Y 410.356,Z 545.804,A -85,B 0,C 180,E1 -10532.945,E2 -10532.945} C_VEL
LIN {X 0,Y 410.285,Z 543.379,A -85,B 0,C 180,E1 -10534.914,E2 -10534.914} C_VEL
LIN {X 0,Y 410.323,Z 539.703,A -85,B 0,C 180,E1 -10536.886,E2 -10536.886} C_VEL
LIN {X 0,Y 410.32,Z 534.678,A -85,B 0,C 180,E1 -10538.868,E2 -10538.868} C_VEL
LIN {X 0,Y 410.588,Z 528.204,A -85,B 0,C 180,E1 -10540.853,E2 -10540.853} C_VEL
LIN {X 0,Y 411.008,Z 520.076,A -85,B 0,C 180,E1 -10542.844,E2 -10542.844} C_VEL
LIN {X 0,Y 411.663,Z 511.419,A -85,B 0,C 180,E1 -10544.585,E2 -10544.585} C_VEL
LIN {X 0,Y 412.424,Z 502.655,A -85,B 0,C 180,E1 -10546.076,E2 -10546.076} C_VEL
LIN {X 0,Y 413.48,Z 492.294,A -85,B 0,C 180,E1 -10547.56,E2 -10547.56} C_VEL
LIN {X 0,Y 414.652,Z 479.939,A -85,B 0,C 180,E1 -10549.043,E2 -10549.043} C_VEL
LIN {X 0,Y 415.883,Z 467.561,A -85,B 0,C 180,E1 -10550.269,E2 -10550.269} C_VEL
LIN {X 0,Y 417.155,Z 454.083,A -85,B 0,C 180,E1 -10551.366,E2 -10551.366} C_VEL
LIN {X 0,Y 418.431,Z 439.44,A -85,B 0,C 180,E1 -10552.316,E2 -10552.316} C_VEL
LIN {X 0,Y 419.412,Z 425.633,A -85,B 0,C 180,E1 -10553.009,E2 -10553.009} C_VEL
LIN {X 0,Y 418.241,Z 412.103,A -85,B 0,C 180,E1 -10553.628,E2 -10553.628} C_VEL
LIN {X 0,Y 416.221,Z 397.263,A -85,B 0,C 180,E1 -10554.171,E2 -10554.171} C_VEL
LIN {X 0,Y 413.884,Z 385.122,A -85,B 0,C 180,E1 -10554.613,E2 -10554.613} C_VEL
LIN {X 0,Y 413.219,Z 381.825,A -85,B 0,C 180,E1 -10554.761,E2 -10554.761} C_VEL
LIN {X 0,Y 414.722,Z 366.68,A -85,B 0,C 180,E1 -10558.327,E2 -10558.327} C_VEL
LIN {X 0,Y 416.556,Z 354.194,A -85,B 0,C 180,E1 -10561.536,E2 -10561.536} C_VEL
LIN {X 0,Y 418.915,Z 342.878,A -85,B 0,C 180,E1 -10564.779,E2 -10564.779} C_VEL
LIN {X 0,Y 420.196,Z 338.238,A -85,B 0,C 180,E1 -10566.236,E2 -10566.236} C_VEL
LIN {X 0,Y 420.207,Z 336.152,A -85,B 0,C 180,E1 -10567.021,E2 -10567.021} C_VEL
LIN {X 0,Y 418.832,Z 330.51,A -85,B 0,C 180,E1 -10569.616,E2 -10569.616} C_VEL
LIN {X 0,Y 417.597,Z 325.91,A -85,B 0,C 180,E1 -10572.314,E2 -10572.314} C_VEL
LIN {X 0,Y 416.542,Z 322.425,A -85,B 0,C 180,E1 -10575.124,E2 -10575.124} C_VEL
LIN {X 0,Y 415.735,Z 320.074,A -85,B 0,C 180,E1 -10578.058,E2 -10578.058} C_VEL
LIN {X 0,Y 415.129,Z 318.762,A -85,B 0,C 180,E1 -10581.215,E2 -10581.215} C_VEL
LIN {X 0,Y 414.714,Z 318.457,A -85,B 0,C 180,E1 -10583.621,E2 -10583.621} C_VEL
LIN {X 0,Y 414.178,Z 318.705,A -85,B 0,C 180,E1 -10586.249,E2 -10586.249} C_VEL
LIN {X 0,Y 413.621,Z 319.552,A -85,B 0,C 180,E1 -10589.353,E2 -10589.353} C_VEL
LIN {X 0,Y 413.208,Z 320.902,A -85,B 0,C 180,E1 -10592.663,E2 -10592.663} C_VEL
LIN {X 0,Y 412.877,Z 322.574,A -85,B 0,C 180,E1 -10595.888,E2 -10595.888} C_VEL
LIN {X 0,Y 412.621,Z 324.497,A -85,B 0,C 180,E1 -10599.042,E2 -10599.042} C_VEL
LIN {X 0,Y 412.503,Z 325.549,A -85,B 0,C 180,E1 -10600.596,E2 -10600.596} C_VEL
LIN {X 0,Y 413.832,Z 328.518,A -85,B 0,C 180,E1 -10600.854,E2 -10600.854} C_VEL
LIN {X 0,Y 418.12,Z 338.245,A -85,B 0,C 180,E1 -10601.75,E2 -10601.75} C_VEL
LIN {X 0,Y 420.188,Z 343.936,A -85,B 0,C 180,E1 -10602.274,E2 -10602.274} C_VEL
LIN {X 0,Y 419.213,Z 356.932,A -85,B 0,C 180,E1 -10603.165,E2 -10603.165} C_VEL
LIN {X 0,Y 418.167,Z 368.451,A -85,B 0,C 180,E1 -10604.151,E2 -10604.151} C_VEL
LIN {X 0,Y 417.181,Z 378.741,A -85,B 0,C 180,E1 -10605.238,E2 -10605.238} C_VEL
LIN {X 0,Y 416.065,Z 389.168,A -85,B 0,C 180,E1 -10606.57,E2 -10606.57} C_VEL
LIN {X 0,Y 415.042,Z 398.446,A -85,B 0,C 180,E1 -10608.028,E2 -10608.028} C_VEL
LIN {X 0,Y 414.165,Z 406.046,A -85,B 0,C 180,E1 -10609.514,E2 -10609.514} C_VEL
LIN {X 0,Y 413.256,Z 412.954,A -85,B 0,C 180,E1 -10611.196,E2 -10611.196} C_VEL
LIN {X 0,Y 412.691,Z 417.672,A -85,B 0,C 180,E1 -10612.662,E2 -10612.662} C_VEL
LIN {X 0,Y 412.065,Z 421.333,A -85,B 0,C 180,E1 -10614.127,E2 -10614.127} C_VEL
LIN {X 0,Y 411.951,Z 423.187,A -85,B 0,C 180,E1 -10615.107,E2 -10615.107} C_VEL
LIN {X 0,Y 411.816,Z 424.593,A -85,B 0,C 180,E1 -10616.086,E2 -10616.086} C_VEL
LIN {X 0,Y 411.377,Z 426.275,A -85,B 0,C 180,E1 -10618.042,E2 -10618.042} C_VEL
LIN {X 0,Y 411.282,Z 426.522,A -85,B 0,C 180,E1 -10619.021,E2 -10619.021} C_VEL
LIN {X 0,Y 411.219,Z 426.342,A -85,B 0,C 180,E1 -10620,E2 -10620} C_VEL
LIN {X 0,Y 411.219,Z 425.76,A -85,B 0,C 180,E1 -10620.979,E2 -10620.979} C_VEL
LIN {X 0,Y 411.052,Z 423.459,A -85,B 0,C 180,E1 -10622.94,E2 -10622.94} C_VEL
LIN {X 0,Y 411.234,Z 420.576,A -85,B 0,C 180,E1 -10624.411,E2 -10624.411} C_VEL
LIN {X 0,Y 411.492,Z 416.699,A -85,B 0,C 180,E1 -10625.882,E2 -10625.882} C_VEL
LIN {X 0,Y 411.814,Z 411.743,A -85,B 0,C 180,E1 -10627.354,E2 -10627.354} C_VEL
LIN {X 0,Y 412.201,Z 404.405,A -85,B 0,C 180,E1 -10629.074,E2 -10629.074} C_VEL
LIN {X 0,Y 412.675,Z 396.55,A -85,B 0,C 180,E1 -10630.549,E2 -10630.549} C_VEL
LIN {X 0,Y 413.196,Z 386.932,A -85,B 0,C 180,E1 -10632.026,E2 -10632.026} C_VEL
LIN {X 0,Y 413.969,Z 376.002,A -85,B 0,C 180,E1 -10633.375,E2 -10633.375} C_VEL
LIN {X 0,Y 414.599,Z 365.106,A -85,B 0,C 180,E1 -10634.48,E2 -10634.48} C_VEL
LIN {X 0,Y 415.181,Z 353.011,A -85,B 0,C 180,E1 -10635.473,E2 -10635.473} C_VEL
LIN {X 0,Y 415.85,Z 338.824,A -85,B 0,C 180,E1 -10636.381,E2 -10636.381} C_VEL
LIN {X 0,Y 415.979,Z 335.309,A -85,B 0,C 180,E1 -10636.565,E2 -10636.565} C_VEL
LIN {X 0,Y 412.309,Z 321.349,A -85,B 0,C 180,E1 -10637.34,E2 -10637.34} C_VEL
LIN {X 0,Y 410.592,Z 314.733,A -85,B 0,C 180,E1 -10637.65,E2 -10637.65} C_VEL
LIN {X 0,Y 410.586,Z 312.096,A -85,B 0,C 180,E1 -10640.02,E2 -10640.02} C_VEL
LIN {X 0,Y 410.62,Z 308.658,A -85,B 0,C 180,E1 -10643.182,E2 -10643.182} C_VEL
LIN {X 0,Y 410.605,Z 305.202,A -85,B 0,C 180,E1 -10646.425,E2 -10646.425} C_VEL
LIN {X 0,Y 410.669,Z 301.687,A -85,B 0,C 180,E1 -10649.755,E2 -10649.755} C_VEL
LIN {X 0,Y 410.708,Z 300.214,A -85,B 0,C 180,E1 -10651.174,E2 -10651.174} C_VEL
LIN {X 0,Y 410.85,Z 299.935,A -85,B 0,C 180,E1 -10653.188,E2 -10653.188} C_VEL
LIN {X 0,Y 411.093,Z 299.905,A -85,B 0,C 180,E1 -10655.539,E2 -10655.539} C_VEL
LIN {X 0,Y 411.206,Z 299.887,A -85,B 0,C 180,E1 -10658.168,E2 -10658.168} C_VEL
LIN {X 0,Y 411.166,Z 299.89,A -85,B 0,C 180,E1 -10661.228,E2 -10661.228} C_VEL
LIN {X 0,Y 411.178,Z 299.89,A -85,B 0,C 180,E1 -10664.49,E2 -10664.49} C_VEL
LIN {X 0,Y 411.184,Z 300.083,A -85,B 0,C 180,E1 -10667.7,E2 -10667.7} C_VEL
LIN {X 0,Y 411.442,Z 302.556,A -85,B 0,C 180,E1 -10669.526,E2 -10669.526} C_VEL
LIN {X 0,Y 411.41,Z 306.005,A -85,B 0,C 180,E1 -10672.049,E2 -10672.049} C_VEL
LIN {X 0,Y 411.33,Z 310.875,A -85,B 0,C 180,E1 -10675.678,E2 -10675.678} C_VEL
LIN {X 0,Y 411.253,Z 315.643,A -85,B 0,C 180,E1 -10679.157,E2 -10679.157} C_VEL
LIN {X 0,Y 411.24,Z 318.848,A -85,B 0,C 180,E1 -10681.411,E2 -10681.411} C_VEL
LIN {X 0,Y 411.239,Z 324.606,A -85,B 0,C 180,E1 -10685.148,E2 -10685.148} C_VEL
LIN {X 0,Y 417.34,Z 340.88,A -85,B 0,C 180,E1 -10685.957,E2 -10685.957} C_VEL
LIN {X 0,Y 421.486,Z 353.93,A -85,B 0,C 180,E1 -10686.718,E2 -10686.718} C_VEL
LIN {X 0,Y 420.655,Z 369.266,A -85,B 0,C 180,E1 -10687.466,E2 -10687.466} C_VEL
LIN {X 0,Y 419.686,Z 383.569,A -85,B 0,C 180,E1 -10688.382,E2 -10688.382} C_VEL
LIN {X 0,Y 418.473,Z 397.239,A -85,B 0,C 180,E1 -10689.477,E2 -10689.477} C_VEL
LIN {X 0,Y 417.19,Z 409.792,A -85,B 0,C 180,E1 -10690.709,E2 -10690.709} C_VEL
LIN {X 0,Y 416.043,Z 421.047,A -85,B 0,C 180,E1 -10692.044,E2 -10692.044} C_VEL
LIN {X 0,Y 414.838,Z 431.479,A -85,B 0,C 180,E1 -10693.514,E2 -10693.514} C_VEL
LIN {X 0,Y 413.609,Z 441.628,A -85,B 0,C 180,E1 -10695.233,E2 -10695.233} C_VEL
LIN {X 0,Y 412.722,Z 450.041,A -85,B 0,C 180,E1 -10696.96,E2 -10696.96} C_VEL
LIN {X 0,Y 411.965,Z 457.035,A -85,B 0,C 180,E1 -10698.686,E2 -10698.686} C_VEL
LIN {X 0,Y 411.298,Z 463.495,A -85,B 0,C 180,E1 -10700.658,E2 -10700.658} C_VEL
LIN {X 0,Y 410.944,Z 467.38,A -85,B 0,C 180,E1 -10702.136,E2 -10702.136} C_VEL
LIN {X 0,Y 410.515,Z 471.449,A -85,B 0,C 180,E1 -10704.104,E2 -10704.104} C_VEL
LIN {X 0,Y 410.466,Z 474.285,A -85,B 0,C 180,E1 -10706.073,E2 -10706.073} C_VEL
LIN {X 0,Y 410.276,Z 476.001,A -85,B 0,C 180,E1 -10708.036,E2 -10708.036} C_VEL
LIN {X 0,Y 410.133,Z 476.603,A -85,B 0,C 180,E1 -10710,E2 -10710} C_VEL
LIN {X 0,Y 410.275,Z 476.043,A -85,B 0,C 180,E1 -10711.963,E2 -10711.963} C_VEL
LIN {X 0,Y 410.44,Z 475.351,A -85,B 0,C 180,E1 -10712.936,E2 -10712.936} C_VEL
LIN {X 0,Y 409.921,Z 474.726,A -85,B 0,C 180,E1 -10713.751,E2 -10713.751} C_VEL
LIN {X 0,Y 407.175,Z 473.422,A -85,B 0,C 180,E1 -10715.072,E2 -10715.072} C_VEL
LIN {X 0,Y 404.808,Z 471.963,A -85,B 0,C 180,E1 -10716.128,E2 -10716.128} C_VEL
LIN {X 0,Y 403.832,Z 470.516,A -85,B 0,C 180,E1 -10716.933,E2 -10716.933} C_VEL
LIN {X 0,Y 403.78,Z 469.954,A -85,B 0,C 180,E1 -10717.202,E2 -10717.202} C_VEL
LIN {X 0,Y 404.141,Z 465.741,A -85,B 0,C 180,E1 -10719.004,E2 -10719.004} C_VEL
LIN {X 0,Y 404.782,Z 459.718,A -85,B 0,C 180,E1 -10721.01,E2 -10721.01} C_VEL
LIN {X 0,Y 405.667,Z 452.131,A -85,B 0,C 180,E1 -10723.016,E2 -10723.016} C_VEL
LIN {X 0,Y 406.542,Z 444.382,A -85,B 0,C 180,E1 -10724.705,E2 -10724.705} C_VEL
LIN {X 0,Y 407.617,Z 435.782,A -85,B 0,C 180,E1 -10726.271,E2 -10726.271} C_VEL
LIN {X 0,Y 408.822,Z 426.014,A -85,B 0,C 180,E1 -10727.766,E2 -10727.766} C_VEL
LIN {X 0,Y 409.968,Z 415.134,A -85,B 0,C 180,E1 -10729.177,E2 -10729.177} C_VEL
LIN {X 0,Y 411.367,Z 402.784,A -85,B 0,C 180,E1 -10730.501,E2 -10730.501} C_VEL
LIN {X 0,Y 412.558,Z 390.21,A -85,B 0,C 180,E1 -10731.616,E2 -10731.616} C_VEL
LIN {X 0,Y 413.702,Z 376.468,A -85,B 0,C 180,E1 -10732.603,E2 -10732.603} C_VEL
LIN {X 0,Y 414.621,Z 362.517,A -85,B 0,C 180,E1 -10733.396,E2 -10733.396} C_VEL
LIN {X 0,Y 414.835,Z 355.141,A -85,B 0,C 180,E1 -10733.748,E2 -10733.748} C_VEL
LIN {X 0,Y 410.186,Z 340.774,A -85,B 0,C 180,E1 -10734.611,E2 -10734.611} C_VEL
LIN {X 0,Y 404.238,Z 325.151,A -85,B 0,C 180,E1 -10735.435,E2 -10735.435} C_VEL
LIN {X 0,Y 404.244,Z 321.158,A -85,B 0,C 180,E1 -10737.996,E2 -10737.996} C_VEL
LIN {X 0,Y 404.273,Z 317.866,A -85,B 0,C 180,E1 -10740.274,E2 -10740.274} C_VEL
LIN {X 0,Y 404.313,Z 312.982,A -85,B 0,C 180,E1 -10743.796,E2 -10743.796} C_VEL
LIN {X 0,Y 404.38,Z 308.093,A -85,B 0,C 180,E1 -10747.466,E2 -10747.466} C_VEL
LIN {X 0,Y 404.446,Z 304.436,A -85,B 0,C 180,E1 -10750.13,E2 -10750.13} C_VEL
LIN {X 0,Y 404.132,Z 300.773,A -85,B 0,C 180,E1 -10752.893,E2 -10752.893} C_VEL
LIN {X 0,Y 404.148,Z 300.771,A -85,B 0,C 180,E1 -10755.926,E2 -10755.926} C_VEL
LIN {X 0,Y 404.118,Z 300.771,A -85,B 0,C 180,E1 -10758.635,E2 -10758.635} C_VEL
LIN {X 0,Y 404.149,Z 300.766,A -85,B 0,C 180,E1 -10761.493,E2 -10761.493} C_VEL
LIN {X 0,Y 404.185,Z 300.765,A -85,B 0,C 180,E1 -10764.984,E2 -10764.984} C_VEL
LIN {X 0,Y 404.142,Z 300.77,A -85,B 0,C 180,E1 -10768.554,E2 -10768.554} C_VEL
LIN {X 0,Y 404.151,Z 300.766,A -85,B 0,C 180,E1 -10770.862,E2 -10770.862} C_VEL
LIN {X 0,Y 404.151,Z 300.761,A -85,B 0,C 180,E1 -10774.723,E2 -10774.723} C_VEL
LIN {X 0,Y 404.17,Z 300.758,A -85,B 0,C 180,E1 -10777.508,E2 -10777.508} C_VEL
LIN {X 0,Y 404.162,Z 300.766,A -85,B 0,C 180,E1 -10780.707,E2 -10780.707} C_VEL
LIN {X 0,Y 404.222,Z 300.75,A -85,B 0,C 180,E1 -10783.848,E2 -10783.848} C_VEL
LIN {X 0,Y 404.283,Z 300.746,A -85,B 0,C 180,E1 -10786.939,E2 -10786.939} C_VEL
LIN {X 0,Y 404.257,Z 300.75,A -85,B 0,C 180,E1 -10789.988,E2 -10789.988} C_VEL
LIN {X 0,Y 404.342,Z 300.736,A -85,B 0,C 180,E1 -10793.011,E2 -10793.011} C_VEL
LIN {X 0,Y 404.27,Z 300.743,A -85,B 0,C 180,E1 -10795.013,E2 -10795.013} C_VEL
LIN {X 0,Y 404.48,Z 300.724,A -85,B 0,C 180,E1 -10798.008,E2 -10798.008} C_VEL
LIN {X 0,Y 404.61,Z 300.695,A -85,B 0,C 180,E1 -10800,E2 -10800} C_VEL
LIN {X 0,Y 404.403,Z 300.735,A -85,B 0,C 180,E1 -10802.988,E2 -10802.988} C_VEL
LIN {X 0,Y 404.382,Z 300.735,A -85,B 0,C 180,E1 -10806.988,E2 -10806.988} C_VEL
LIN {X 0,Y 404.258,Z 300.745,A -85,B 0,C 180,E1 -10810.012,E2 -10810.012} C_VEL
LIN {X 0,Y 404.266,Z 300.752,A -85,B 0,C 180,E1 -10813.211,E2 -10813.211} C_VEL
LIN {X 0,Y 404.216,Z 300.748,A -85,B 0,C 180,E1 -10817.007,E2 -10817.007} C_VEL
LIN {X 0,Y 404.164,Z 300.761,A -85,B 0,C 180,E1 -10820.351,E2 -10820.351} C_VEL
LIN {X 0,Y 404.156,Z 300.767,A -85,B 0,C 180,E1 -10823.575,E2 -10823.575} C_VEL
LIN {X 0,Y 404.129,Z 300.76,A -85,B 0,C 180,E1 -10826.882,E2 -10826.882} C_VEL
LIN {X 0,Y 404.143,Z 300.77,A -85,B 0,C 180,E1 -10830.285,E2 -10830.285} C_VEL
LIN {X 0,Y 404.144,Z 300.769,A -85,B 0,C 180,E1 -10833.812,E2 -10833.812} C_VEL
LIN {X 0,Y 404.134,Z 300.771,A -85,B 0,C 180,E1 -10836.875,E2 -10836.875} C_VEL
LIN {X 0,Y 404.147,Z 300.769,A -85,B 0,C 180,E1 -10840.08,E2 -10840.08} C_VEL
LIN {X 0,Y 404.161,Z 300.912,A -85,B 0,C 180,E1 -10842.922,E2 -10842.922} C_VEL
LIN {X 0,Y 406.608,Z 310.948,A -85,B 0,C 180,E1 -10846.261,E2 -10846.261} C_VEL
LIN {X 0,Y 409.439,Z 322.317,A -85,B 0,C 180,E1 -10849.803,E2 -10849.803} C_VEL
LIN {X 0,Y 412.314,Z 334.184,A -85,B 0,C 180,E1 -10853.238,E2 -10853.238} C_VEL
LIN {X 0,Y 411.983,Z 338.135,A -85,B 0,C 180,E1 -10854.249,E2 -10854.249} C_VEL
LIN {X 0,Y 410.025,Z 351.373,A -85,B 0,C 180,E1 -10857.478,E2 -10857.478} C_VEL
LIN {X 0,Y 408.226,Z 365.721,A -85,B 0,C 180,E1 -10860.899,E2 -10860.899} C_VEL
LIN {X 0,Y 406.714,Z 380.784,A -85,B 0,C 180,E1 -10864.406,E2 -10864.406} C_VEL
LIN {X 0,Y 406.474,Z 383.079,A -85,B 0,C 180,E1 -10864.935,E2 -10864.935} C_VEL
LIN {X 0,Y 410.165,Z 403.861,A -85,B 0,C 180,E1 -10865.625,E2 -10865.625} C_VEL
LIN {X 0,Y 411.905,Z 416.967,A -85,B 0,C 180,E1 -10866.181,E2 -10866.181} C_VEL
LIN {X 0,Y 412.684,Z 427.281,A -85,B 0,C 180,E1 -10866.7,E2 -10866.7} C_VEL
LIN {X 0,Y 411.608,Z 441.266,A -85,B 0,C 180,E1 -10867.448,E2 -10867.448} C_VEL
LIN {X 0,Y 410.283,Z 455.137,A -85,B 0,C 180,E1 -10868.39,E2 -10868.39} C_VEL
LIN {X 0,Y 408.944,Z 468.316,A -85,B 0,C 180,E1 -10869.503,E2 -10869.503} C_VEL
LIN {X 0,Y 407.699,Z 480.469,A -85,B 0,C 180,E1 -10870.751,E2 -10870.751} C_VEL
LIN {X 0,Y 406.485,Z 492.393,A -85,B 0,C 180,E1 -10872.226,E2 -10872.226} C_VEL
LIN {X 0,Y 405.517,Z 502.073,A -85,B 0,C 180,E1 -10873.643,E2 -10873.643} C_VEL
LIN {X 0,Y 404.572,Z 512.199,A -85,B 0,C 180,E1 -10875.411,E2 -10875.411} C_VEL
LIN {X 0,Y 403.819,Z 520.733,A -85,B 0,C 180,E1 -10877.208,E2 -10877.208} C_VEL
LIN {X 0,Y 403.507,Z 527.597,A -85,B 0,C 180,E1 -10878.955,E2 -10878.955} C_VEL
LIN {X 0,Y 403.225,Z 534.076,A -85,B 0,C 180,E1 -10880.975,E2 -10880.975} C_VEL
LIN {X 0,Y 403.189,Z 539.094,A -85,B 0,C 180,E1 -10882.992,E2 -10882.992} C_VEL
LIN {X 0,Y 403.157,Z 542.765,A -85,B 0,C 180,E1 -10885,E2 -10885} C_VEL
LIN {X 0,Y 403.271,Z 545.193,A -85,B 0,C 180,E1 -10887.003,E2 -10887.003} C_VEL
LIN {X 0,Y 403.218,Z 546.404,A -85,B 0,C 180,E1 -10889.002,E2 -10889.002} C_VEL
LIN {X 0,Y 403.217,Z 546.404,A -85,B 0,C 180,E1 -10890.999,E2 -10890.999} C_VEL
LIN {X 0,Y 403.284,Z 545.195,A -85,B 0,C 180,E1 -10892.997,E2 -10892.997} C_VEL
LIN {X 0,Y 403.209,Z 542.768,A -85,B 0,C 180,E1 -10895,E2 -10895} C_VEL
LIN {X 0,Y 403.215,Z 539.087,A -85,B 0,C 180,E1 -10897.008,E2 -10897.008} C_VEL
LIN {X 0,Y 403.251,Z 534.063,A -85,B 0,C 180,E1 -10899.025,E2 -10899.025} C_VEL
LIN {X 0,Y 403.529,Z 527.587,A -85,B 0,C 180,E1 -10901.045,E2 -10901.045} C_VEL
LIN {X 0,Y 403.995,Z 519.459,A -85,B 0,C 180,E1 -10903.071,E2 -10903.071} C_VEL
LIN {X 0,Y 404.676,Z 510.8,A -85,B 0,C 180,E1 -10904.843,E2 -10904.843} C_VEL
LIN {X 0,Y 405.523,Z 502.04,A -85,B 0,C 180,E1 -10906.357,E2 -10906.357} C_VEL
LIN {X 0,Y 406.648,Z 491.682,A -85,B 0,C 180,E1 -10907.865,E2 -10907.865} C_VEL
LIN {X 0,Y 407.738,Z 480.416,A -85,B 0,C 180,E1 -10909.248,E2 -10909.248} C_VEL
LIN {X 0,Y 409.017,Z 468.255,A -85,B 0,C 180,E1 -10910.494,E2 -10910.494} C_VEL
LIN {X 0,Y 410.328,Z 455.07,A -85,B 0,C 180,E1 -10911.608,E2 -10911.608} C_VEL
LIN {X 0,Y 411.619,Z 441.211,A -85,B 0,C 180,E1 -10912.549,E2 -10912.549} C_VEL
LIN {X 0,Y 412.67,Z 427.122,A -85,B 0,C 180,E1 -10913.301,E2 -10913.301} C_VEL
LIN {X 0,Y 411.536,Z 411.52,A -85,B 0,C 180,E1 -10914.037,E2 -10914.037} C_VEL
LIN {X 0,Y 409.295,Z 396.223,A -85,B 0,C 180,E1 -10914.617,E2 -10914.617} C_VEL
LIN {X 0,Y 406.412,Z 380.774,A -85,B 0,C 180,E1 -10915.341,E2 -10915.341} C_VEL
LIN {X 0,Y 408.156,Z 365.379,A -85,B 0,C 180,E1 -10919.107,E2 -10919.107} C_VEL
LIN {X 0,Y 409.98,Z 354.21,A -85,B 0,C 180,E1 -10922.101,E2 -10922.101} C_VEL
LIN {X 0,Y 412.559,Z 343.184,A -85,B 0,C 180,E1 -10925.394,E2 -10925.394} C_VEL
LIN {X 0,Y 413.5,Z 339.811,A -85,B 0,C 180,E1 -10926.504,E2 -10926.504} C_VEL
LIN {X 0,Y 413.11,Z 336.735,A -85,B 0,C 180,E1 -10927.767,E2 -10927.767} C_VEL
LIN {X 0,Y 411.782,Z 331.354,A -85,B 0,C 180,E1 -10930.433,E2 -10930.433} C_VEL
LIN {X 0,Y 410.534,Z 327.07,A -85,B 0,C 180,E1 -10933.218,E2 -10933.218} C_VEL
LIN {X 0,Y 409.552,Z 323.884,A -85,B 0,C 180,E1 -10936.115,E2 -10936.115} C_VEL
LIN {X 0,Y 409.077,Z 322.481,A -85,B 0,C 180,E1 -10937.931,E2 -10937.931} C_VEL
LIN {X 0,Y 408.444,Z 321.121,A -85,B 0,C 180,E1 -10940.742,E2 -10940.742} C_VEL
LIN {X 0,Y 408.077,Z 320.634,A -85,B 0,C 180,E1 -10942.931,E2 -10942.931} C_VEL
LIN {X 0,Y 407.436,Z 320.684,A -85,B 0,C 180,E1 -10945.891,E2 -10945.891} C_VEL
LIN {X 0,Y 406.871,Z 321.305,A -85,B 0,C 180,E1 -10948.789,E2 -10948.789} C_VEL
LIN {X 0,Y 406.4,Z 322.507,A -85,B 0,C 180,E1 -10952.166,E2 -10952.166} C_VEL
LIN {X 0,Y 406.037,Z 324.083,A -85,B 0,C 180,E1 -10955.455,E2 -10955.455} C_VEL
LIN {X 0,Y 405.756,Z 325.935,A -85,B 0,C 180,E1 -10958.67,E2 -10958.67} C_VEL
LIN {X 0,Y 405.706,Z 326.986,A -85,B 0,C 180,E1 -10960.02,E2 -10960.02} C_VEL
LIN {X 0,Y 412.32,Z 341.78,A -85,B 0,C 180,E1 -10961.467,E2 -10961.467} C_VEL
LIN {X 0,Y 413.869,Z 346.906,A -85,B 0,C 180,E1 -10961.951,E2 -10961.951} C_VEL
LIN {X 0,Y 412.715,Z 359.902,A -85,B 0,C 180,E1 -10962.892,E2 -10962.892} C_VEL
LIN {X 0,Y 411.529,Z 372.184,A -85,B 0,C 180,E1 -10964.015,E2 -10964.015} C_VEL
LIN {X 0,Y 410.49,Z 382.038,A -85,B 0,C 180,E1 -10965.119,E2 -10965.119} C_VEL
LIN {X 0,Y 409.432,Z 391.17,A -85,B 0,C 180,E1 -10966.348,E2 -10966.348} C_VEL
LIN {X 0,Y 408.31,Z 400.208,A -85,B 0,C 180,E1 -10967.828,E2 -10967.828} C_VEL
LIN {X 0,Y 407.339,Z 407.98,A -85,B 0,C 180,E1 -10969.399,E2 -10969.399} C_VEL
LIN {X 0,Y 406.412,Z 414.509,A -85,B 0,C 180,E1 -10971.046,E2 -10971.046} C_VEL
LIN {X 0,Y 405.791,Z 419.106,A -85,B 0,C 180,E1 -10972.537,E2 -10972.537} C_VEL
LIN {X 0,Y 405.153,Z 422.667,A -85,B 0,C 180,E1 -10974.026,E2 -10974.026} C_VEL
LIN {X 0,Y 404.997,Z 424.471,A -85,B 0,C 180,E1 -10975.023,E2 -10975.023} C_VEL
LIN {X 0,Y 404.866,Z 425.836,A -85,B 0,C 180,E1 -10976.019,E2 -10976.019} C_VEL
LIN {X 0,Y 404.4,Z 427.443,A -85,B 0,C 180,E1 -10978.008,E2 -10978.008} C_VEL
LIN {X 0,Y 404.294,Z 427.64,A -85,B 0,C 180,E1 -10979.004,E2 -10979.004} C_VEL
LIN {X 0,Y 404.197,Z 426.79,A -85,B 0,C 180,E1 -10980.996,E2 -10980.996} C_VEL
LIN {X 0,Y 404.082,Z 425.801,A -85,B 0,C 180,E1 -10981.994,E2 -10981.994} C_VEL
LIN {X 0,Y 404.025,Z 424.401,A -85,B 0,C 180,E1 -10982.991,E2 -10982.991} C_VEL
LIN {X 0,Y 404.22,Z 421.459,A -85,B 0,C 180,E1 -10984.487,E2 -10984.487} C_VEL
LIN {X 0,Y 404.498,Z 417.506,A -85,B 0,C 180,E1 -10985.984,E2 -10985.984} C_VEL
LIN {X 0,Y 404.823,Z 412.475,A -85,B 0,C 180,E1 -10987.482,E2 -10987.482} C_VEL
LIN {X 0,Y 405.16,Z 406.224,A -85,B 0,C 180,E1 -10988.982,E2 -10988.982} C_VEL
LIN {X 0,Y 405.629,Z 398.519,A -85,B 0,C 180,E1 -10990.482,E2 -10990.482} C_VEL
LIN {X 0,Y 406.162,Z 389.094,A -85,B 0,C 180,E1 -10991.984,E2 -10991.984} C_VEL
LIN {X 0,Y 406.922,Z 378.488,A -85,B 0,C 180,E1 -10993.356,E2 -10993.356} C_VEL
LIN {X 0,Y 407.639,Z 366.591,A -85,B 0,C 180,E1 -10994.605,E2 -10994.605} C_VEL
LIN {X 0,Y 408.228,Z 355.001,A -85,B 0,C 180,E1 -10995.594,E2 -10995.594} C_VEL
LIN {X 0,Y 408.896,Z 342.01,A -85,B 0,C 180,E1 -10996.465,E2 -10996.465} C_VEL
LIN {X 0,Y 409.046,Z 336.553,A -85,B 0,C 180,E1 -10996.773,E2 -10996.773} C_VEL
LIN {X 0,Y 405.465,Z 322.604,A -85,B 0,C 180,E1 -10997.573,E2 -10997.573} C_VEL
LIN {X 0,Y 403.547,Z 315.273,A -85,B 0,C 180,E1 -10997.93,E2 -10997.93} C_VEL
LIN {X 0,Y 403.522,Z 312.55,A -85,B 0,C 180,E1 -11000.386,E2 -11000.386} C_VEL
LIN {X 0,Y 403.573,Z 309.06,A -85,B 0,C 180,E1 -11003.612,E2 -11003.612} C_VEL
LIN {X 0,Y 403.586,Z 305.519,A -85,B 0,C 180,E1 -11006.921,E2 -11006.921} C_VEL
LIN {X 0,Y 403.625,Z 301.956,A -85,B 0,C 180,E1 -11010.328,E2 -11010.328} C_VEL
LIN {X 0,Y 403.668,Z 300.831,A -85,B 0,C 180,E1 -11011.487,E2 -11011.487} C_VEL
LIN {X 0,Y 404.043,Z 300.783,A -85,B 0,C 180,E1 -11015.161,E2 -11015.161} C_VEL
LIN {X 0,Y 404.156,Z 300.767,A -85,B 0,C 180,E1 -11018.508,E2 -11018.508} C_VEL
LIN {X 0,Y 404.125,Z 300.766,A -85,B 0,C 180,E1 -11021.6,E2 -11021.6} C_VEL
LIN {X 0,Y 404.147,Z 300.766,A -85,B 0,C 180,E1 -11024.522,E2 -11024.522} C_VEL
LIN {X 0,Y 404.145,Z 300.801,A -85,B 0,C 180,E1 -11027.296,E2 -11027.296} C_VEL
LIN {X 0,Y 404.431,Z 302.666,A -85,B 0,C 180,E1 -11028.673,E2 -11028.673} C_VEL
LIN {X 0,Y 404.42,Z 306.412,A -85,B 0,C 180,E1 -11031.445,E2 -11031.445} C_VEL
LIN {X 0,Y 404.349,Z 310.889,A -85,B 0,C 180,E1 -11034.777,E2 -11034.777} C_VEL
LIN {X 0,Y 404.277,Z 315.846,A -85,B 0,C 180,E1 -11038.411,E2 -11038.411} C_VEL
LIN {X 0,Y 404.263,Z 319.327,A -85,B 0,C 180,E1 -11040.871,E2 -11040.871} C_VEL
LIN {X 0,Y 404.233,Z 324.463,A -85,B 0,C 180,E1 -11044.237,E2 -11044.237} C_VEL
LIN {X 0,Y 404.248,Z 325.201,A -85,B 0,C 180,E1 -11044.694,E2 -11044.694} C_VEL
LIN {X 0,Y 410.433,Z 341.463,A -85,B 0,C 180,E1 -11045.526,E2 -11045.526} C_VEL
LIN {X 0,Y 414.935,Z 355.457,A -85,B 0,C 180,E1 -11046.371,E2 -11046.371} C_VEL
LIN {X 0,Y 414.141,Z 369.853,A -85,B 0,C 180,E1 -11047.092,E2 -11047.092} C_VEL
LIN {X 0,Y 413.118,Z 384.163,A -85,B 0,C 180,E1 -11048.021,E2 -11048.021} C_VEL
LIN {X 0,Y 411.862,Z 397.837,A -85,B 0,C 180,E1 -11049.132,E2 -11049.132} C_VEL
LIN {X 0,Y 410.498,Z 410.646,A -85,B 0,C 180,E1 -11050.41,E2 -11050.41} C_VEL
LIN {X 0,Y 409.325,Z 421.65,A -85,B 0,C 180,E1 -11051.739,E2 -11051.739} C_VEL
LIN {X 0,Y 408.046,Z 432.086,A -85,B 0,C 180,E1 -11053.232,E2 -11053.232} C_VEL
LIN {X 0,Y 406.751,Z 442.237,A -85,B 0,C 180,E1 -11054.979,E2 -11054.979} C_VEL
LIN {X 0,Y 405.822,Z 450.65,A -85,B 0,C 180,E1 -11056.734,E2 -11056.734} C_VEL
LIN {X 0,Y 405.019,Z 457.644,A -85,B 0,C 180,E1 -11058.489,E2 -11058.489} C_VEL
LIN {X 0,Y 404.311,Z 464.104,A -85,B 0,C 180,E1 -11060.495,E2 -11060.495} C_VEL
LIN {X 0,Y 403.916,Z 467.99,A -85,B 0,C 180,E1 -11061.998,E2 -11061.998} C_VEL
LIN {X 0,Y 403.475,Z 472.058,A -85,B 0,C 180,E1 -11064.001,E2 -11064.001} C_VEL
LIN {X 0,Y 403.414,Z 474.894,A -85,B 0,C 180,E1 -11066.004,E2 -11066.004} C_VEL
LIN {X 0,Y 403.229,Z 476.607,A -85,B 0,C 180,E1 -11068.002,E2 -11068.002} C_VEL
LIN {X 0,Y 403.078,Z 477.21,A -85,B 0,C 180,E1 -11070,E2 -11070} C_VEL
LIN {X 0,Y 403.229,Z 476.649,A -85,B 0,C 180,E1 -11071.997,E2 -11071.997} C_VEL
LIN {X 0,Y 403.406,Z 474.992,A -85,B 0,C 180,E1 -11073.996,E2 -11073.996} C_VEL
LIN {X 0,Y 403.477,Z 472.219,A -85,B 0,C 180,E1 -11075.999,E2 -11075.999} C_VEL
LIN {X 0,Y 403.78,Z 469.954,A -85,B 0,C 180,E1 -11077.202,E2 -11077.202} C_VEL
LIN {X 0,Y 403.238,Z 468.318,A -85,B 0,C 180,E1 -11078.003,E2 -11078.003} C_VEL
LIN {X 0,Y 400.674,Z 465.436,A -85,B 0,C 180,E1 -11079.309,E2 -11079.309} C_VEL
LIN {X 0,Y 398.592,Z 462.866,A -85,B 0,C 180,E1 -11080.347,E2 -11080.347} C_VEL
LIN {X 0,Y 397.863,Z 460.586,A -85,B 0,C 180,E1 -11081.125,E2 -11081.125} C_VEL
LIN {X 0,Y 397.893,Z 459.72,A -85,B 0,C 180,E1 -11081.381,E2 -11081.381} C_VEL
LIN {X 0,Y 398.763,Z 452.736,A -85,B 0,C 180,E1 -11083.245,E2 -11083.245} C_VEL
LIN {X 0,Y 399.678,Z 445.145,A -85,B 0,C 180,E1 -11084.932,E2 -11084.932} C_VEL
LIN {X 0,Y 400.827,Z 436.383,A -85,B 0,C 180,E1 -11086.554,E2 -11086.554} C_VEL
LIN {X 0,Y 402.088,Z 426.612,A -85,B 0,C 180,E1 -11088.074,E2 -11088.074} C_VEL
LIN {X 0,Y 403.416,Z 414.586,A -85,B 0,C 180,E1 -11089.648,E2 -11089.648} C_VEL
LIN {X 0,Y 404.887,Z 402.124,A -85,B 0,C 180,E1 -11090.978,E2 -11090.978} C_VEL
LIN {X 0,Y 406.149,Z 389.265,A -85,B 0,C 180,E1 -11092.108,E2 -11092.108} C_VEL
LIN {X 0,Y 407.352,Z 375.131,A -85,B 0,C 180,E1 -11093.11,E2 -11093.11} C_VEL
LIN {X 0,Y 408.342,Z 359.473,A -85,B 0,C 180,E1 -11093.972,E2 -11093.972} C_VEL
LIN {X 0,Y 408.235,Z 356.566,A -85,B 0,C 180,E1 -11094.116,E2 -11094.116} C_VEL
LIN {X 0,Y 403.573,Z 342.164,A -85,B 0,C 180,E1 -11095.014,E2 -11095.014} C_VEL
LIN {X 0,Y 398.043,Z 328.122,A -85,B 0,C 180,E1 -11095.779,E2 -11095.779} C_VEL
LIN {X 0,Y 397.254,Z 325.729,A -85,B 0,C 180,E1 -11095.918,E2 -11095.918} C_VEL
LIN {X 0,Y 397.257,Z 321.666,A -85,B 0,C 180,E1 -11098.533,E2 -11098.533} C_VEL
LIN {X 0,Y 397.281,Z 318.31,A -85,B 0,C 180,E1 -11100.865,E2 -11100.865} C_VEL
LIN {X 0,Y 397.329,Z 313.336,A -85,B 0,C 180,E1 -11104.473,E2 -11104.473} C_VEL
LIN {X 0,Y 397.417,Z 308.31,A -85,B 0,C 180,E1 -11108.239,E2 -11108.239} C_VEL
LIN {X 0,Y 397.412,Z 304.733,A -85,B 0,C 180,E1 -11110.868,E2 -11110.868} C_VEL
LIN {X 0,Y 397.09,Z 301.65,A -85,B 0,C 180,E1 -11113.171,E2 -11113.171} C_VEL
LIN {X 0,Y 397.102,Z 301.649,A -85,B 0,C 180,E1 -11116.521,E2 -11116.521} C_VEL
LIN {X 0,Y 397.112,Z 301.642,A -85,B 0,C 180,E1 -11120.422,E2 -11120.422} C_VEL
LIN {X 0,Y 397.108,Z 301.645,A -85,B 0,C 180,E1 -11124.265,E2 -11124.265} C_VEL
LIN {X 0,Y 397.115,Z 301.639,A -85,B 0,C 180,E1 -11126.727,E2 -11126.727} C_VEL
LIN {X 0,Y 397.117,Z 301.637,A -85,B 0,C 180,E1 -11130.295,E2 -11130.295} C_VEL
LIN {X 0,Y 397.079,Z 301.64,A -85,B 0,C 180,E1 -11133.738,E2 -11133.738} C_VEL
LIN {X 0,Y 397.108,Z 301.64,A -85,B 0,C 180,E1 -11137.085,E2 -11137.085} C_VEL
LIN {X 0,Y 397.146,Z 301.642,A -85,B 0,C 180,E1 -11140.353,E2 -11140.353} C_VEL
LIN {X 0,Y 397.167,Z 301.626,A -85,B 0,C 180,E1 -11143.553,E2 -11143.553} C_VEL
LIN {X 0,Y 397.229,Z 301.628,A -85,B 0,C 180,E1 -11146.703,E2 -11146.703} C_VEL
LIN {X 0,Y 397.216,Z 301.625,A -85,B 0,C 180,E1 -11149.809,E2 -11149.809} C_VEL
LIN {X 0,Y 397.294,Z 301.615,A -85,B 0,C 180,E1 -11152.887,E2 -11152.887} C_VEL
LIN {X 0,Y 397.24,Z 301.617,A -85,B 0,C 180,E1 -11154.925,E2 -11154.925} C_VEL
LIN {X 0,Y 397.449,Z 301.6,A -85,B 0,C 180,E1 -11157.973,E2 -11157.973} C_VEL
LIN {X 0,Y 397.579,Z 301.57,A -85,B 0,C 180,E1 -11160,E2 -11160} C_VEL
LIN {X 0,Y 397.337,Z 301.616,A -85,B 0,C 180,E1 -11163.042,E2 -11163.042} C_VEL
LIN {X 0,Y 397.346,Z 301.605,A -85,B 0,C 180,E1 -11166.092,E2 -11166.092} C_VEL
LIN {X 0,Y 397.236,Z 301.625,A -85,B 0,C 180,E1 -11169.162,E2 -11169.162} C_VEL
LIN {X 0,Y 397.219,Z 301.625,A -85,B 0,C 180,E1 -11172.258,E2 -11172.258} C_VEL
LIN {X 0,Y 397.177,Z 301.627,A -85,B 0,C 180,E1 -11175.392,E2 -11175.392} C_VEL
LIN {X 0,Y 397.158,Z 301.639,A -85,B 0,C 180,E1 -11178.574,E2 -11178.574} C_VEL
LIN {X 0,Y 397.095,Z 301.634,A -85,B 0,C 180,E1 -11181.818,E2 -11181.818} C_VEL
LIN {X 0,Y 397.106,Z 301.643,A -85,B 0,C 180,E1 -11185.135,E2 -11185.135} C_VEL
LIN {X 0,Y 397.078,Z 301.65,A -85,B 0,C 180,E1 -11188.547,E2 -11188.547} C_VEL
LIN {X 0,Y 397.081,Z 301.65,A -85,B 0,C 180,E1 -11191.837,E2 -11191.837} C_VEL
LIN {X 0,Y 397.124,Z 301.642,A -85,B 0,C 180,E1 -11194.493,E2 -11194.493} C_VEL
LIN {X 0,Y 397.097,Z 301.649,A -85,B 0,C 180,E1 -11198.276,E2 -11198.276} C_VEL
LIN {X 0,Y 397.088,Z 301.646,A -85,B 0,C 180,E1 -11200.909,E2 -11200.909} C_VEL
LIN {X 0,Y 397.093,Z 301.794,A -85,B 0,C 180,E1 -11202.35,E2 -11202.35} C_VEL
LIN {X 0,Y 399.403,Z 311.169,A -85,B 0,C 180,E1 -11205.572,E2 -11205.572} C_VEL
LIN {X 0,Y 401.849,Z 321.106,A -85,B 0,C 180,E1 -11208.767,E2 -11208.767} C_VEL
LIN {X 0,Y 404.488,Z 332.005,A -85,B 0,C 180,E1 -11212.055,E2 -11212.055} C_VEL
LIN {X 0,Y 405.473,Z 336.807,A -85,B 0,C 180,E1 -11213.421,E2 -11213.421} C_VEL
LIN {X 0,Y 403.451,Z 350.011,A -85,B 0,C 180,E1 -11216.735,E2 -11216.735} C_VEL
LIN {X 0,Y 401.491,Z 364.826,A -85,B 0,C 180,E1 -11220.363,E2 -11220.363} C_VEL
LIN {X 0,Y 399.814,Z 379.761,A -85,B 0,C 180,E1 -11223.931,E2 -11223.931} C_VEL
LIN {X 0,Y 399.632,Z 382.189,A -85,B 0,C 180,E1 -11224.468,E2 -11224.468} C_VEL
LIN {X 0,Y 403.334,Z 402.934,A -85,B 0,C 180,E1 -11225.173,E2 -11225.173} C_VEL
LIN {X 0,Y 405.162,Z 416.638,A -85,B 0,C 180,E1 -11225.771,E2 -11225.771} C_VEL
LIN {X 0,Y 405.994,Z 428.507,A -85,B 0,C 180,E1 -11226.387,E2 -11226.387} C_VEL
LIN {X 0,Y 404.811,Z 442.82,A -85,B 0,C 180,E1 -11227.193,E2 -11227.193} C_VEL
LIN {X 0,Y 403.462,Z 456.134,A -85,B 0,C 180,E1 -11228.14,E2 -11228.14} C_VEL
LIN {X 0,Y 402.082,Z 469.018,A -85,B 0,C 180,E1 -11229.271,E2 -11229.271} C_VEL
LIN {X 0,Y 400.789,Z 480.943,A -85,B 0,C 180,E1 -11230.539,E2 -11230.539} C_VEL
LIN {X 0,Y 399.558,Z 492.433,A -85,B 0,C 180,E1 -11232.002,E2 -11232.002} C_VEL
LIN {X 0,Y 398.436,Z 502.988,A -85,B 0,C 180,E1 -11233.607,E2 -11233.607} C_VEL
LIN {X 0,Y 397.465,Z 512.848,A -85,B 0,C 180,E1 -11235.406,E2 -11235.406} C_VEL
LIN {X 0,Y 396.744,Z 520.736,A -85,B 0,C 180,E1 -11237.124,E2 -11237.124} C_VEL
LIN {X 0,Y 396.457,Z 526.982,A -85,B 0,C 180,E1 -11238.756,E2 -11238.756} C_VEL
LIN {X 0,Y 396.126,Z 533.46,A -85,B 0,C 180,E1 -11240.812,E2 -11240.812} C_VEL
LIN {X 0,Y 396.094,Z 538.481,A -85,B 0,C 180,E1 -11242.865,E2 -11242.865} C_VEL
LIN {X 0,Y 396.088,Z 542.155,A -85,B 0,C 180,E1 -11244.91,E2 -11244.91} C_VEL
LIN {X 0,Y 396.199,Z 544.584,A -85,B 0,C 180,E1 -11246.95,E2 -11246.95} C_VEL
LIN {X 0,Y 396.16,Z 545.797,A -85,B 0,C 180,E1 -11248.984,E2 -11248.984} C_VEL
LIN {X 0,Y 396.159,Z 545.797,A -85,B 0,C 180,E1 -11251.017,E2 -11251.017} C_VEL
LIN {X 0,Y 396.213,Z 544.586,A -85,B 0,C 180,E1 -11253.051,E2 -11253.051} C_VEL
LIN {X 0,Y 396.137,Z 542.158,A -85,B 0,C 180,E1 -11255.089,E2 -11255.089} C_VEL
LIN {X 0,Y 396.112,Z 538.471,A -85,B 0,C 180,E1 -11257.135,E2 -11257.135} C_VEL
LIN {X 0,Y 396.174,Z 533.447,A -85,B 0,C 180,E1 -11259.187,E2 -11259.187} C_VEL
LIN {X 0,Y 396.479,Z 526.97,A -85,B 0,C 180,E1 -11261.244,E2 -11261.244} C_VEL
LIN {X 0,Y 397.001,Z 518.843,A -85,B 0,C 180,E1 -11263.305,E2 -11263.305} C_VEL
LIN {X 0,Y 397.703,Z 510.181,A -85,B 0,C 180,E1 -11265.109,E2 -11265.109} C_VEL
LIN {X 0,Y 398.621,Z 501.425,A -85,B 0,C 180,E1 -11266.649,E2 -11266.649} C_VEL
LIN {X 0,Y 399.82,Z 490.866,A -85,B 0,C 180,E1 -11268.21,E2 -11268.21} C_VEL
LIN {X 0,Y 400.951,Z 479.803,A -85,B 0,C 180,E1 -11269.587,E2 -11269.587} C_VEL
LIN {X 0,Y 402.281,Z 467.646,A -85,B 0,C 180,E1 -11270.853,E2 -11270.853} C_VEL
LIN {X 0,Y 403.701,Z 454.47,A -85,B 0,C 180,E1 -11271.981,E2 -11271.981} C_VEL
LIN {X 0,Y 405,Z 440.886,A -85,B 0,C 180,E1 -11272.92,E2 -11272.92} C_VEL
LIN {X 0,Y 405.988,Z 426.32,A -85,B 0,C 180,E1 -11273.719,E2 -11273.719} C_VEL
LIN {X 0,Y 404.802,Z 410.932,A -85,B 0,C 180,E1 -11274.463,E2 -11274.463} C_VEL
LIN {X 0,Y 402.847,Z 396.575,A -85,B 0,C 180,E1 -11275.088,E2 -11275.088} C_VEL
LIN {X 0,Y 400.301,Z 382.973,A -85,B 0,C 180,E1 -11275.775,E2 -11275.775} C_VEL
LIN {X 0,Y 399.673,Z 379.769,A -85,B 0,C 180,E1 -11275.944,E2 -11275.944} C_VEL
LIN {X 0,Y 401.463,Z 365.209,A -85,B 0,C 180,E1 -11279.64,E2 -11279.64} C_VEL
LIN {X 0,Y 403.674,Z 353.135,A -85,B 0,C 180,E1 -11283.024,E2 -11283.024} C_VEL
LIN {X 0,Y 406.203,Z 343.513,A -85,B 0,C 180,E1 -11286.034,E2 -11286.034} C_VEL
LIN {X 0,Y 406.688,Z 341.881,A -85,B 0,C 180,E1 -11286.598,E2 -11286.598} C_VEL
LIN {X 0,Y 406.352,Z 338.81,A -85,B 0,C 180,E1 -11287.878,E2 -11287.878} C_VEL
LIN {X 0,Y 405.182,Z 334.056,A -85,B 0,C 180,E1 -11290.254,E2 -11290.254} C_VEL
LIN {X 0,Y 403.933,Z 329.698,A -85,B 0,C 180,E1 -11293.05,E2 -11293.05} C_VEL
LIN {X 0,Y 402.975,Z 326.565,A -85,B 0,C 180,E1 -11295.764,E2 -11295.764} C_VEL
LIN {X 0,Y 402.151,Z 324.321,A -85,B 0,C 180,E1 -11298.718,E2 -11298.718} C_VEL
LIN {X 0,Y 401.683,Z 323.29,A -85,B 0,C 180,E1 -11300.96,E2 -11300.96} C_VEL
LIN {X 0,Y 401.153,Z 322.716,A -85,B 0,C 180,E1 -11303.698,E2 -11303.698} C_VEL
LIN {X 0,Y 400.38,Z 322.899,A -85,B 0,C 180,E1 -11307.033,E2 -11307.033} C_VEL
LIN {X 0,Y 399.743,Z 323.776,A -85,B 0,C 180,E1 -11310.51,E2 -11310.51} C_VEL
LIN {X 0,Y 399.337,Z 325.109,A -85,B 0,C 180,E1 -11313.898,E2 -11313.898} C_VEL
LIN {X 0,Y 399.017,Z 326.783,A -85,B 0,C 180,E1 -11317.202,E2 -11317.202} C_VEL
LIN {X 0,Y 398.793,Z 328.073,A -85,B 0,C 180,E1 -11319.362,E2 -11319.362} C_VEL
LIN {X 0,Y 400.188,Z 331.111,A -85,B 0,C 180,E1 -11319.676,E2 -11319.676} C_VEL
LIN {X 0,Y 405.665,Z 343.063,A -85,B 0,C 180,E1 -11320.944,E2 -11320.944} C_VEL
LIN {X 0,Y 407.593,Z 348.443,A -85,B 0,C 180,E1 -11321.505,E2 -11321.505} C_VEL
LIN {X 0,Y 406.418,Z 361.693,A -85,B 0,C 180,E1 -11322.499,E2 -11322.499} C_VEL
LIN {X 0,Y 404.998,Z 374.784,A -85,B 0,C 180,E1 -11323.751,E2 -11323.751} C_VEL
LIN {X 0,Y 403.657,Z 386.218,A -85,B 0,C 180,E1 -11325.119,E2 -11325.119} C_VEL
LIN {X 0,Y 402.416,Z 396.382,A -85,B 0,C 180,E1 -11326.62,E2 -11326.62} C_VEL
LIN {X 0,Y 401.213,Z 404.671,A -85,B 0,C 180,E1 -11328.122,E2 -11328.122} C_VEL
LIN {X 0,Y 400.097,Z 412.382,A -85,B 0,C 180,E1 -11329.883,E2 -11329.883} C_VEL
LIN {X 0,Y 399.38,Z 417.659,A -85,B 0,C 180,E1 -11331.398,E2 -11331.398} C_VEL
LIN {X 0,Y 398.583,Z 421.848,A -85,B 0,C 180,E1 -11332.91,E2 -11332.91} C_VEL
LIN {X 0,Y 398.235,Z 424.059,A -85,B 0,C 180,E1 -11333.922,E2 -11333.922} C_VEL
LIN {X 0,Y 398.044,Z 425.78,A -85,B 0,C 180,E1 -11334.935,E2 -11334.935} C_VEL
LIN {X 0,Y 397.91,Z 427.085,A -85,B 0,C 180,E1 -11335.949,E2 -11335.949} C_VEL
LIN {X 0,Y 397.419,Z 428.609,A -85,B 0,C 180,E1 -11337.973,E2 -11337.973} C_VEL
LIN {X 0,Y 397.303,Z 428.748,A -85,B 0,C 180,E1 -11338.987,E2 -11338.987} C_VEL
LIN {X 0,Y 397.183,Z 428.486,A -85,B 0,C 180,E1 -11340,E2 -11340} C_VEL
LIN {X 0,Y 397.174,Z 427.818,A -85,B 0,C 180,E1 -11341.014,E2 -11341.014} C_VEL
LIN {X 0,Y 397.058,Z 426.781,A -85,B 0,C 180,E1 -11342.029,E2 -11342.029} C_VEL
LIN {X 0,Y 396.995,Z 425.321,A -85,B 0,C 180,E1 -11343.044,E2 -11343.044} C_VEL
LIN {X 0,Y 397.207,Z 422.306,A -85,B 0,C 180,E1 -11344.567,E2 -11344.567} C_VEL
LIN {X 0,Y 397.503,Z 418.281,A -85,B 0,C 180,E1 -11346.09,E2 -11346.09} C_VEL
LIN {X 0,Y 397.831,Z 413.172,A -85,B 0,C 180,E1 -11347.614,E2 -11347.614} C_VEL
LIN {X 0,Y 398.25,Z 405.619,A -85,B 0,C 180,E1 -11349.395,E2 -11349.395} C_VEL
LIN {X 0,Y 398.765,Z 397.592,A -85,B 0,C 180,E1 -11350.922,E2 -11350.922} C_VEL
LIN {X 0,Y 399.219,Z 389.527,A -85,B 0,C 180,E1 -11352.196,E2 -11352.196} C_VEL
LIN {X 0,Y 400.019,Z 378.782,A -85,B 0,C 180,E1 -11353.591,E2 -11353.591} C_VEL
LIN {X 0,Y 400.788,Z 366.772,A -85,B 0,C 180,E1 -11354.86,E2 -11354.86} C_VEL
LIN {X 0,Y 401.395,Z 354.822,A -85,B 0,C 180,E1 -11355.881,E2 -11355.881} C_VEL
LIN {X 0,Y 402.118,Z 340.594,A -85,B 0,C 180,E1 -11356.829,E2 -11356.829} C_VEL
LIN {X 0,Y 402.099,Z 337.478,A -85,B 0,C 180,E1 -11357.007,E2 -11357.007} C_VEL
LIN {X 0,Y 398.47,Z 323.441,A -85,B 0,C 180,E1 -11357.837,E2 -11357.837} C_VEL
LIN {X 0,Y 396.49,Z 315.833,A -85,B 0,C 180,E1 -11358.204,E2 -11358.204} C_VEL
LIN {X 0,Y 396.489,Z 313.001,A -85,B 0,C 180,E1 -11360.764,E2 -11360.764} C_VEL
LIN {X 0,Y 396.507,Z 309.428,A -85,B 0,C 180,E1 -11364.059,E2 -11364.059} C_VEL
LIN {X 0,Y 396.526,Z 305.691,A -85,B 0,C 180,E1 -11367.6,E2 -11367.6} C_VEL
LIN {X 0,Y 396.593,Z 302.213,A -85,B 0,C 180,E1 -11370.925,E2 -11370.925} C_VEL
LIN {X 0,Y 396.655,Z 301.704,A -85,B 0,C 180,E1 -11372.11,E2 -11372.11} C_VEL
LIN {X 0,Y 397.006,Z 301.66,A -85,B 0,C 180,E1 -11375.48,E2 -11375.48} C_VEL
LIN {X 0,Y 397.132,Z 301.641,A -85,B 0,C 180,E1 -11378.861,E2 -11378.861} C_VEL
LIN {X 0,Y 397.071,Z 301.645,A -85,B 0,C 180,E1 -11382.267,E2 -11382.267} C_VEL
LIN {X 0,Y 397.088,Z 301.645,A -85,B 0,C 180,E1 -11385.069,E2 -11385.069} C_VEL
LIN {X 0,Y 397.099,Z 301.8,A -85,B 0,C 180,E1 -11387.047,E2 -11387.047} C_VEL
LIN {X 0,Y 397.467,Z 305.046,A -85,B 0,C 180,E1 -11389.493,E2 -11389.493} C_VEL
LIN {X 0,Y 397.4,Z 309.825,A -85,B 0,C 180,E1 -11393.037,E2 -11393.037} C_VEL
LIN {X 0,Y 397.319,Z 314.118,A -85,B 0,C 180,E1 -11396.239,E2 -11396.239} C_VEL
LIN {X 0,Y 397.304,Z 319.485,A -85,B 0,C 180,E1 -11400.086,E2 -11400.086} C_VEL
LIN {X 0,Y 397.237,Z 323.233,A -85,B 0,C 180,E1 -11402.613,E2 -11402.613} C_VEL
LIN {X 0,Y 397.276,Z 325.727,A -85,B 0,C 180,E1 -11404.194,E2 -11404.194} C_VEL
LIN {X 0,Y 404.123,Z 343.72,A -85,B 0,C 180,E1 -11405.173,E2 -11405.173} C_VEL
LIN {X 0,Y 408.35,Z 356.907,A -85,B 0,C 180,E1 -11406.007,E2 -11406.007} C_VEL
LIN {X 0,Y 407.565,Z 371.525,A -85,B 0,C 180,E1 -11406.768,E2 -11406.768} C_VEL
LIN {X 0,Y 406.562,Z 384.758,A -85,B 0,C 180,E1 -11407.647,E2 -11407.647} C_VEL
LIN {X 0,Y 405.259,Z 398.436,A -85,B 0,C 180,E1 -11408.776,E2 -11408.776} C_VEL
LIN {X 0,Y 403.989,Z 410.148,A -85,B 0,C 180,E1 -11409.953,E2 -11409.953} C_VEL
LIN {X 0,Y 402.6,Z 422.255,A -85,B 0,C 180,E1 -11411.423,E2 -11411.423} C_VEL
LIN {X 0,Y 401.253,Z 432.694,A -85,B 0,C 180,E1 -11412.939,E2 -11412.939} C_VEL
LIN {X 0,Y 400.116,Z 441.531,A -85,B 0,C 180,E1 -11414.462,E2 -11414.462} C_VEL
LIN {X 0,Y 399.072,Z 450.179,A -85,B 0,C 180,E1 -11416.246,E2 -11416.246} C_VEL
LIN {X 0,Y 398.077,Z 458.253,A -85,B 0,C 180,E1 -11418.285,E2 -11418.285} C_VEL
LIN {X 0,Y 397.334,Z 464.712,A -85,B 0,C 180,E1 -11420.326,E2 -11420.326} C_VEL
LIN {X 0,Y 396.907,Z 468.599,A -85,B 0,C 180,E1 -11421.856,E2 -11421.856} C_VEL
LIN {X 0,Y 396.439,Z 472.667,A -85,B 0,C 180,E1 -11423.894,E2 -11423.894} C_VEL
LIN {X 0,Y 396.363,Z 475.502,A -85,B 0,C 180,E1 -11425.933,E2 -11425.933} C_VEL
LIN {X 0,Y 396.184,Z 477.214,A -85,B 0,C 180,E1 -11427.967,E2 -11427.967} C_VEL
LIN {X 0,Y 396.024,Z 477.816,A -85,B 0,C 180,E1 -11430,E2 -11430} C_VEL
LIN {X 0,Y 396.183,Z 477.255,A -85,B 0,C 180,E1 -11432.033,E2 -11432.033} C_VEL
LIN {X 0,Y 396.356,Z 475.599,A -85,B 0,C 180,E1 -11434.067,E2 -11434.067} C_VEL
LIN {X 0,Y 396.441,Z 472.826,A -85,B 0,C 180,E1 -11436.106,E2 -11436.106} C_VEL
LIN {X 0,Y 396.905,Z 468.828,A -85,B 0,C 180,E1 -11438.143,E2 -11438.143} C_VEL
LIN {X 0,Y 397.456,Z 463.519,A -85,B 0,C 180,E1 -11440.185,E2 -11440.185} C_VEL
LIN {X 0,Y 397.893,Z 459.72,A -85,B 0,C 180,E1 -11441.381,E2 -11441.381} C_VEL
LIN {X 0,Y 397.585,Z 457.169,A -85,B 0,C 180,E1 -11442.147,E2 -11442.147} C_VEL
LIN {X 0,Y 395.358,Z 452.925,A -85,B 0,C 180,E1 -11443.405,E2 -11443.405} C_VEL
LIN {X 0,Y 393.175,Z 448.247,A -85,B 0,C 180,E1 -11444.638,E2 -11444.638} C_VEL
LIN {X 0,Y 392.934,Z 444.959,A -85,B 0,C 180,E1 -11445.354,E2 -11445.354} C_VEL
LIN {X 0,Y 394.234,Z 435.456,A -85,B 0,C 180,E1 -11447.106,E2 -11447.106} C_VEL
LIN {X 0,Y 395.605,Z 425.446,A -85,B 0,C 180,E1 -11448.649,E2 -11448.649} C_VEL
LIN {X 0,Y 396.933,Z 413.737,A -85,B 0,C 180,E1 -11450.164,E2 -11450.164} C_VEL
LIN {X 0,Y 398.47,Z 401.423,A -85,B 0,C 180,E1 -11451.468,E2 -11451.468} C_VEL
LIN {X 0,Y 399.813,Z 388.284,A -85,B 0,C 180,E1 -11452.614,E2 -11452.614} C_VEL
